// Datatypes/Structs/_TcVnKeyPoint
{attribute 'linkalways'} 
{attribute 'no_explicit_call' := 'This FB is a CLASS and must be accessed using methods or properties'}
{attribute 'enable_dynamic_creation'}
FUNCTION_BLOCK _TcVnKeyPoint EXTENDS StructuredDatatypeBase
VAR
	localData : TcVnKeyPoint;
	activeData : REFERENCE TO TcVnKeyPoint REF= localData;
    _aPoint : _TcVnPoint2_REAL();
    _fDiameter : _REAL(localdata.fDiameter);
    _fAngle : _REAL(localdata.fAngle);
    _fResponse : _REAL(localdata.fResponse);
    _nOctave : _DINT(localdata.nOctave);
    _nClassId : _DINT(localdata.nClassId);
END_VAR

PROPERTY PUBLIC Address : PVOID
GET
Address := ADR(activeData);
END_GET
END_PROPERTY

METHOD PUBLIC ClearReference
VAR_INPUT
END_VAR
activeData REF= localData;
SetMemberReference();
END_METHOD

PROPERTY PUBLIC Size : UDINT
GET
Size := SIZEOF(activeData);
END_GET
END_PROPERTY

METHOD FB_init : BOOL
VAR_INPUT
	bInitRetains : BOOL; // if TRUE, the retain variables are initialized (warm start / cold start)
	bInCopyCode : BOOL;  // if TRUE, the instance afterwards gets moved into the copy code (online change)
END_VAR
SetMemberReference();
AddMember('aPoint', _aPoint);
AddMember('fDiameter', _fDiameter);
AddMember('fAngle', _fAngle);
AddMember('fResponse', _fResponse);
AddMember('nOctave', _nOctave);
AddMember('nClassId', _nClassId);
END_METHOD

METHOD PROTECTED SetMemberReference
VAR_INPUT
END_VAR
_aPoint.MakeReferenceTo(activeData.aPoint);
_fDiameter.MakeReferenceTo(activeData.fDiameter);
_fAngle.MakeReferenceTo(activeData.fAngle);
_fResponse.MakeReferenceTo(activeData.fResponse);
_nOctave.MakeReferenceTo(activeData.nOctave);
_nClassId.MakeReferenceTo(activeData.nClassId);
END_METHOD

METHOD PUBLIC Clone : I_Datatype
VAR
    pClone : POINTER TO _TcVnKeyPoint;
END_VAR
pClone := __NEW(_TcVnKeyPoint());
pClone^.Value := Value;
Clone := pClone^;
END_METHOD

PROPERTY PUBLIC Identifier : T_MAXSTRING
GET
Identifier := 'TcVnKeyPoint';
END_GET
END_PROPERTY

METHOD PUBLIC MakeReferenceTo
VAR_INPUT
	ReferenceTarget : REFERENCE TO TcVnKeyPoint;
END_VAR
activeData REF= ReferenceTarget;
SetMemberReference();
END_METHOD

METHOD TryMakeReferenceTo : BOOL
VAR_INPUT
	Target : I_Datatype;
END_VAR
VAR
	pTargetData : POINTER TO TcVnKeyPoint;
END_VAR
IF NOT IsEquivalentTo(Target) THEN
	RETURN;
END_IF

pTargetData := Target.Address;
activeData REF= pTargetData^;
SetMemberReference();
TryMakeReferenceTo := TRUE;
END_METHOD

PROPERTY PUBLIC Value : REFERENCE TO TcVnKeyPoint
GET
Value REF= activeData;
END_GET
END_PROPERTY

PROPERTY PUBLIC aPoint : REFERENCE TO _TcVnPoint2_REAL
GET
aPoint REF= _aPoint;
END_GET
END_PROPERTY

PROPERTY PUBLIC fAngle : REFERENCE TO _REAL
GET
fAngle REF= _fAngle;
END_GET
END_PROPERTY

PROPERTY PUBLIC fDiameter : REFERENCE TO _REAL
GET
fDiameter REF= _fDiameter;
END_GET
END_PROPERTY

PROPERTY PUBLIC fResponse : REFERENCE TO _REAL
GET
fResponse REF= _fResponse;
END_GET
END_PROPERTY

PROPERTY PUBLIC nClassId : REFERENCE TO _DINT
GET
nClassId REF= _nClassId;
END_GET
END_PROPERTY

PROPERTY PUBLIC nOctave : REFERENCE TO _DINT
GET
nOctave REF= _nOctave;
END_GET
END_PROPERTY

END_FUNCTION_BLOCK

// Datatypes/Structs/_TcVnRotatedRectangle
{attribute 'linkalways'} 
{attribute 'no_explicit_call' := 'This FB is a CLASS and must be accessed using methods or properties'}
{attribute 'enable_dynamic_creation'}
FUNCTION_BLOCK _TcVnRotatedRectangle EXTENDS StructuredDatatypeBase
VAR
	localData : TcVnRotatedRectangle;
	activeData : REFERENCE TO TcVnRotatedRectangle REF= localData;
    _aCenter : _TcVnPoint2_REAL();
    _stSize : _TcVnSize2_REAL();
    _fAngle : _REAL(localdata.fAngle);
END_VAR

PROPERTY PUBLIC Address : PVOID
GET
Address := ADR(activeData);
END_GET
END_PROPERTY

METHOD PUBLIC ClearReference
VAR_INPUT
END_VAR
activeData REF= localData;
SetMemberReference();
END_METHOD

PROPERTY PUBLIC Size : UDINT
GET
Size := SIZEOF(activeData);
END_GET
END_PROPERTY

METHOD FB_init : BOOL
VAR_INPUT
	bInitRetains : BOOL; // if TRUE, the retain variables are initialized (warm start / cold start)
	bInCopyCode : BOOL;  // if TRUE, the instance afterwards gets moved into the copy code (online change)
END_VAR
SetMemberReference();
AddMember('aCenter', _aCenter);
AddMember('stSize', _stSize);
AddMember('fAngle', _fAngle);
END_METHOD

METHOD PROTECTED SetMemberReference
VAR_INPUT
END_VAR
_aCenter.MakeReferenceTo(activeData.aCenter);
_stsize.MakeReferenceTo(activeData.stSize);
_fAngle.MakeReferenceTo(activeData.fAngle);
END_METHOD

METHOD PUBLIC Clone : I_Datatype
VAR
    pClone : POINTER TO _TcVnRotatedRectangle;
END_VAR
pClone := __NEW(_TcVnRotatedRectangle());
pClone^.Value := Value;
Clone := pClone^;
END_METHOD

PROPERTY PUBLIC Identifier : T_MAXSTRING
GET
Identifier := 'TcVnRotatedRectangle';
END_GET
END_PROPERTY

METHOD PUBLIC MakeReferenceTo
VAR_INPUT
	ReferenceTarget : REFERENCE TO TcVnRotatedRectangle;
END_VAR
activeData REF= ReferenceTarget;
SetMemberReference();
END_METHOD

METHOD TryMakeReferenceTo : BOOL
VAR_INPUT
	Target : I_Datatype;
END_VAR
VAR
	pTargetData : POINTER TO TcVnRotatedRectangle;
END_VAR
IF NOT IsEquivalentTo(Target) THEN
	RETURN;
END_IF

pTargetData := Target.Address;
activeData REF= pTargetData^;
SetMemberReference();
TryMakeReferenceTo := TRUE;
END_METHOD

PROPERTY PUBLIC Value : REFERENCE TO TcVnRotatedRectangle
GET
Value REF= activeData;
END_GET
END_PROPERTY

PROPERTY PUBLIC aCenter : REFERENCE TO _TcVnPoint2_REAL
GET
aCenter REF= _aCenter;
END_GET
END_PROPERTY

PROPERTY PUBLIC fAngle : REFERENCE TO _REAL
GET
fAngle REF= _fAngle;
END_GET
END_PROPERTY

PROPERTY PUBLIC stSize : REFERENCE TO _TcVnSize2_REAL
GET
stSize REF= _stSize;
END_GET
END_PROPERTY

END_FUNCTION_BLOCK

// Datatypes/Structs/_TcVnSize2_REAL
{attribute 'linkalways'} 
{attribute 'no_explicit_call' := 'This FB is a CLASS and must be accessed using methods or properties'}
{attribute 'enable_dynamic_creation'}
FUNCTION_BLOCK _TcVnSize2_REAL EXTENDS StructuredDatatypeBase
VAR
	localData : TcVnSize2_REAL;
	activeData : REFERENCE TO TcVnSize2_REAL REF= localData;
    _fWidth : _REAL(localdata.fWidth);
    _fHeight : _REAL(localdata.fHeight);
END_VAR

PROPERTY PUBLIC Address : PVOID
GET
Address := ADR(activeData);
END_GET
END_PROPERTY

METHOD PUBLIC ClearReference
VAR_INPUT
END_VAR
activeData REF= localData;
SetMemberReference();
END_METHOD

PROPERTY PUBLIC Size : UDINT
GET
Size := SIZEOF(activeData);
END_GET
END_PROPERTY

METHOD FB_init : BOOL
VAR_INPUT
	bInitRetains : BOOL; // if TRUE, the retain variables are initialized (warm start / cold start)
	bInCopyCode : BOOL;  // if TRUE, the instance afterwards gets moved into the copy code (online change)
END_VAR
SetMemberReference();
AddMember('fWidth', _fWidth);
AddMember('fHeight', _fHeight);
END_METHOD

METHOD PROTECTED SetMemberReference
VAR_INPUT
END_VAR
_fWidth.MakeReferenceTo(activeData.fWidth);
_fHeight.MakeReferenceTo(activeData.fHeight);
END_METHOD

METHOD PUBLIC Clone : I_Datatype
VAR
    pClone : POINTER TO _TcVnSize2_REAL;
END_VAR
pClone := __NEW(_TcVnSize2_REAL());
pClone^.Value := Value;
Clone := pClone^;
END_METHOD

PROPERTY PUBLIC Identifier : T_MAXSTRING
GET
Identifier := 'TcVnSize2_REAL';
END_GET
END_PROPERTY

METHOD PUBLIC MakeReferenceTo
VAR_INPUT
	ReferenceTarget : REFERENCE TO TcVnSize2_REAL;
END_VAR
activeData REF= ReferenceTarget;
SetMemberReference();
END_METHOD

METHOD TryMakeReferenceTo : BOOL
VAR_INPUT
	Target : I_Datatype;
END_VAR
VAR
	pTargetData : POINTER TO TcVnSize2_REAL;
END_VAR
IF NOT IsEquivalentTo(Target) THEN
	RETURN;
END_IF

pTargetData := Target.Address;
activeData REF= pTargetData^;
SetMemberReference();
TryMakeReferenceTo := TRUE;
END_METHOD

PROPERTY PUBLIC Value : REFERENCE TO TcVnSize2_REAL
GET
Value REF= activeData;
END_GET
END_PROPERTY

PROPERTY PUBLIC fHeight : REFERENCE TO _REAL
GET
fHeight REF= _fHeight;
END_GET
END_PROPERTY

PROPERTY PUBLIC fWidth : REFERENCE TO _REAL
GET
fWidth REF= _fWidth;
END_GET
END_PROPERTY

END_FUNCTION_BLOCK

// Datatypes/Interfaces/Containers/Iterators/ITcVnBidirectionalIterator/_ITcVnBidirectionalIterator
{attribute 'linkalways'} 
{attribute 'no_explicit_call' := 'This FB is a CLASS and must be accessed using methods or properties'}
{attribute 'enable_dynamic_creation'}
FUNCTION_BLOCK _ITcVnBidirectionalIterator EXTENDS InterfaceDatatypeBase IMPLEMENTS I_InterfaceDatatype_ITcVnBidirectionalIterator
VAR
	localData : ITcVnBidirectionalIterator;
	activeData : REFERENCE TO ITcVnBidirectionalIterator REF= localData;
END_VAR

PROPERTY PUBLIC Address : PVOID
GET
Address := ADR(activeData);
END_GET
END_PROPERTY

METHOD PUBLIC ClearReference
VAR_INPUT
END_VAR
activeData REF= localData;
END_METHOD

PROPERTY PUBLIC Size : UDINT
GET
Size := SIZEOF(activeData);
END_GET
END_PROPERTY

METHOD FB_exit : BOOL
VAR_INPUT
	bInCopyCode : BOOL; // if TRUE, the exit method is called for exiting an instance that is copied afterwards (online change).
END_VAR
IF bInCopyCode THEN
	RETURN;
END_IF

TryTcReleaseLocal();
END_METHOD

METHOD PUBLIC TryTcReleaseLocal : BOOL
VAR_INPUT
END_VAR
IF localData = 0 THEN
	RETURN;
END_IF

IF localData.TcRelease() = 0 THEN
	localData := 0;
END_IF

TryTcReleaseLocal := TRUE;
END_METHOD

METHOD PUBLIC Clone : I_Datatype
VAR
    pClone : POINTER TO _ITcVnBidirectionalIterator;
END_VAR
pClone := __NEW(_ITcVnBidirectionalIterator);
Clone := pClone^;
END_METHOD

PROPERTY PUBLIC Identifier : T_MAXSTRING
GET
Identifier := 'ITcVnBidirectionalIterator';
END_GET
END_PROPERTY

METHOD PUBLIC MakeReferenceTo
VAR_INPUT
	ReferenceTarget : REFERENCE TO ITcVnBidirectionalIterator;
END_VAR
activeData REF= ReferenceTarget;
END_METHOD

METHOD PUBLIC SerializeWith
VAR_INPUT
	Serializer : I_Serializer;
END_VAR
Serializer.AddNull();
END_METHOD

METHOD TryDeserializeFrom : BOOL
VAR_INPUT
	Deserializer : I_Deserializer;
	Feedback : I_DeserializerFeedback;
END_VAR
VAR
END_VAR
// not implemented.
END_METHOD

METHOD TryMakeReferenceTo : BOOL
VAR_INPUT
	Target : I_Datatype;
END_VAR
VAR
	pTargetData : POINTER TO ITcVnBidirectionalIterator;
END_VAR
IF NOT IsEquivalentTo(Target) THEN
	RETURN;
END_IF

pTargetData := Target.Address;
activeData REF= pTargetData^;
TryMakeReferenceTo := TRUE;
END_METHOD

PROPERTY PUBLIC Value : REFERENCE TO ITcVnBidirectionalIterator
GET
Value REF= activeData;
END_GET
END_PROPERTY

PROPERTY PUBLIC IsValid : BOOL
GET
IsValid := activeData <> 0;
END_GET
END_PROPERTY

METHOD PUBLIC TryCheckIfBegin : BOOL
VAR_INPUT
	Result : REFERENCE TO BOOL;
END_VAR
Result := FALSE;

IF NOT IsValid THEN
	RETURN;
END_IF

IF activeData.CheckIfBegin() = S_OK THEN
    Result := TRUE;
END_IF

TryCheckIfBegin := TRUE;
END_METHOD

METHOD PUBLIC TryCheckIfEnd : BOOL
VAR_INPUT
	Result : REFERENCE TO BOOL;
END_VAR
Result := FALSE;

IF NOT IsValid THEN
	RETURN;
END_IF

IF activeData.CheckIfEnd() = S_OK THEN
    Result := TRUE;
END_IF

TryCheckIfEnd := TRUE;
END_METHOD

METHOD PUBLIC TryCopyContentFrom : BOOL
VAR_INPUT
	Source : I_InterfaceDatatype;
END_VAR
// currently un-copyable
END_METHOD

METHOD PUBLIC TryGetValueSize : BOOL
VAR_INPUT
	Destination : REFERENCE TO ULINT;
END_VAR
IF NOT IsValid THEN
	RETURN;
END_IF

TryGetValueSize := SUCCEEDED(activeData.GetValueSize(Destination));
END_METHOD

METHOD PUBLIC TryGetValueTypeGuid : BOOL
VAR_INPUT
	Destination : REFERENCE TO GUID;
END_VAR
IF NOT IsValid THEN
	RETURN;
END_IF

TryGetValueTypeGuid := SUCCEEDED(activeData.GetValueTypeGuid(Destination));
END_METHOD

METHOD PUBLIC TryTcAddRef : BOOL
VAR_INPUT
END_VAR
IF activeData = 0 THEN
	RETURN;
END_IF

IF activeData.TcAddRef() = 0 THEN
	activeData := 0;
END_IF

TryTcAddRef := TRUE;
END_METHOD

METHOD PUBLIC TryTcRelease : BOOL
VAR_INPUT
END_VAR
IF activeData = 0 THEN
	RETURN;
END_IF

IF activeData.TcRelease() = 0 THEN
	activeData := 0;
END_IF

TryTcRelease := TRUE;
END_METHOD

END_FUNCTION_BLOCK

// Datatypes/Interfaces/Containers/Iterators/ITcVnBidirectionalIterator/I_InterfaceDatatype_ITcVnBidirectionalIterator
INTERFACE I_InterfaceDatatype_ITcVnBidirectionalIterator EXTENDS I_InterfaceDatatype

PROPERTY PUBLIC Value : REFERENCE TO ITcVnBidirectionalIterator
GET
END_GET
END_PROPERTY

END_INTERFACE

// Datatypes/Interfaces/Images/ITcVnDisplayableImage/_ITcVnDisplayableImage
{attribute 'linkalways'} 
{attribute 'no_explicit_call' := 'This FB is a CLASS and must be accessed using methods or properties'}
{attribute 'enable_dynamic_creation'}
FUNCTION_BLOCK _ITcVnDisplayableImage EXTENDS InterfaceDatatypeBase IMPLEMENTS I_InterfaceDatatype_ITcVnDisplayableImage
VAR
	localData : ITcVnDisplayableImage;
	activeData : REFERENCE TO ITcVnDisplayableImage REF= localData;
END_VAR

PROPERTY PUBLIC Address : PVOID
GET
Address := ADR(activeData);
END_GET
END_PROPERTY

METHOD PUBLIC ClearReference
VAR_INPUT
END_VAR
activeData REF= localData;
END_METHOD

PROPERTY PUBLIC Size : UDINT
GET
Size := SIZEOF(activeData);
END_GET
END_PROPERTY

METHOD FB_exit : BOOL
VAR_INPUT
	bInCopyCode : BOOL; // if TRUE, the exit method is called for exiting an instance that is copied afterwards (online change).
END_VAR
IF bInCopyCode THEN
	RETURN;
END_IF

TryTcReleaseLocal();
END_METHOD

METHOD PUBLIC TryTcReleaseLocal : BOOL
VAR_INPUT
END_VAR
IF localData = 0 THEN
	RETURN;
END_IF

IF localData.TcRelease() = 0 THEN
	localData := 0;
END_IF

TryTcReleaseLocal := TRUE;
END_METHOD

METHOD PUBLIC Clone : I_Datatype
VAR
    pClone : POINTER TO _ITcVnDisplayableImage;
END_VAR
pClone := __NEW(_ITcVnDisplayableImage);
Clone := pClone^;
END_METHOD

PROPERTY PUBLIC Identifier : T_MAXSTRING
GET
Identifier := 'ITcVnDisplayableImage';
END_GET
END_PROPERTY

METHOD PUBLIC MakeReferenceTo
VAR_INPUT
	ReferenceTarget : REFERENCE TO ITcVnDisplayableImage;
END_VAR
activeData REF= ReferenceTarget;
END_METHOD

METHOD PUBLIC SerializeWith
VAR_INPUT
	Serializer : I_Serializer;
END_VAR
// not possible to serialize the data.
Serializer.AddNull();
END_METHOD

METHOD TryMakeReferenceTo : BOOL
VAR_INPUT
	Target : I_Datatype;
END_VAR
VAR
	pTargetData : POINTER TO ITcVnDisplayableImage;
END_VAR
IF NOT IsEquivalentTo(Target) THEN
	RETURN;
END_IF

pTargetData := Target.Address;
activeData REF= pTargetData^;
TryMakeReferenceTo := TRUE;
END_METHOD

PROPERTY PUBLIC Value : REFERENCE TO ITcVnDisplayableImage
GET
Value REF= activeData;
END_GET
END_PROPERTY

PROPERTY PUBLIC IsValid : BOOL
GET
IsValid := activeData <> 0;
END_GET
END_PROPERTY

METHOD PUBLIC TryCopyContentFrom : BOOL
VAR_INPUT
	Source : I_InterfaceDatatype;
END_VAR
// not possible to copy the data, so this will always fail
END_METHOD

METHOD TryDeserializeFrom : BOOL
VAR_INPUT
	Deserializer : I_Deserializer;
	Feedback : I_DeserializerFeedback;
END_VAR
// not possible to deserialize from data.
TryDeserializeFrom := TRUE;
END_METHOD

METHOD PUBLIC TryTcAddRef : BOOL
VAR_INPUT
END_VAR
IF activeData = 0 THEN
	RETURN;
END_IF

IF activeData.TcAddRef() = 0 THEN
	activeData := 0;
END_IF

TryTcAddRef := TRUE;
END_METHOD

METHOD PUBLIC TryTcRelease : BOOL
VAR_INPUT
END_VAR
IF activeData = 0 THEN
	RETURN;
END_IF

IF activeData.TcRelease() = 0 THEN
	activeData := 0;
END_IF

TryTcRelease := TRUE;
END_METHOD

END_FUNCTION_BLOCK

// Datatypes/Interfaces/Images/ITcVnDisplayableImage/I_InterfaceDatatype_ITcVnDisplayableImage
INTERFACE I_InterfaceDatatype_ITcVnDisplayableImage EXTENDS I_InterfaceDatatype

PROPERTY PUBLIC Value : REFERENCE TO ITcVnDisplayableImage
GET
END_GET
END_PROPERTY

END_INTERFACE

// Datatypes/Structs/_GVCP_ADDRESS_VALUE_PAIR
{attribute 'linkalways'}
{attribute 'no_explicit_call' := 'This FB is a CLASS and must be accessed using methods or properties'}
{attribute 'enable_dynamic_creation'}
FUNCTION_BLOCK _GVCP_ADDRESS_VALUE_PAIR EXTENDS StructuredDatatypeBase
VAR
    localData : GVCP_ADDRESS_VALUE_PAIR;
    activeData : REFERENCE TO GVCP_ADDRESS_VALUE_PAIR REF= localData;
    _nAddress : _GVCP_REGISTER_ADDRESS(0);
    _nValue : _GVCP_REGISTER_VALUE(0);
END_VAR

PROPERTY PUBLIC Address : PVOID
GET
Address := ADR(activeData);
END_GET
END_PROPERTY

METHOD PUBLIC ClearReference
VAR_INPUT
END_VAR
activeData REF= localData;
SetMemberReference();
END_METHOD

PROPERTY PUBLIC Size : UDINT
GET
Size := SIZEOF(activeData);
END_GET
END_PROPERTY

METHOD FB_init : BOOL
VAR_INPUT
	bInitRetains : BOOL; // if TRUE, the retain variables are initialized (warm start / cold start)
	bInCopyCode : BOOL;  // if TRUE, the instance afterwards gets moved into the copy code (online change)
END_VAR
SetMemberReference();
AddMember('nAddress', _nAddress);
AddMember('nValue', _nValue);
END_METHOD

METHOD PROTECTED SetMemberReference
VAR_INPUT
END_VAR
_nAddress.MakeReferenceTo(activeData.nAddress);
_nValue.MakeReferenceTo(activeData.nValue);
END_METHOD

METHOD PUBLIC Clone : I_Datatype
VAR
    pClone : POINTER TO _GVCP_ADDRESS_VALUE_PAIR;
END_VAR
pClone := __NEW(_GVCP_ADDRESS_VALUE_PAIR);
IF pClone = 0 THEN
    RETURN;
END_IF
pClone^.TryCopyFrom(THIS^);
Clone := pClone^;
END_METHOD

PROPERTY PUBLIC Identifier : T_MAXSTRING
GET
Identifier := 'GVCP_ADDRESS_VALUE_PAIR';
END_GET
END_PROPERTY

METHOD PUBLIC MakeReferenceTo
VAR_INPUT
	ReferenceTarget : REFERENCE TO GVCP_ADDRESS_VALUE_PAIR;
END_VAR
activeData REF= ReferenceTarget;
SetMemberReference();
END_METHOD

METHOD TryMakeReferenceTo : BOOL
VAR_INPUT
	Target : I_Datatype;
END_VAR
VAR
	pTargetData : POINTER TO GVCP_ADDRESS_VALUE_PAIR;
END_VAR
IF NOT IsEquivalentTo(Target) THEN
	RETURN;
END_IF

pTargetData := Target.Address;
activeData REF= pTargetData^;
SetMemberReference();
TryMakeReferenceTo := TRUE;
END_METHOD

PROPERTY PUBLIC Value : REFERENCE TO GVCP_ADDRESS_VALUE_PAIR
GET
Value REF= activeData;
END_GET
END_PROPERTY

PROPERTY PUBLIC nAddress : REFERENCE TO _GVCP_REGISTER_ADDRESS
GET
nAddress REF= _nAddress;
END_GET
END_PROPERTY

PROPERTY PUBLIC nValue : REFERENCE TO _GVCP_REGISTER_VALUE
GET
nValue REF= _nValue;
END_GET
END_PROPERTY

END_FUNCTION_BLOCK

// Datatypes/Structs/_GVSP_IMAGE_INFO
{attribute 'linkalways'} 
{attribute 'no_explicit_call' := 'This FB is a CLASS and must be accessed using methods or properties'}
{attribute 'enable_dynamic_creation'}
FUNCTION_BLOCK _GVSP_IMAGE_INFO EXTENDS StructuredDatatypeBase
VAR
	localData : GVSP_IMAGE_INFO;
	activeData : REFERENCE TO GVSP_IMAGE_INFO REF= localData;
    _CameraIpAddress : _UDINT(localdata.CameraIpAddress);
    _LocalIpAddress : _UDINT(localdata.LocalIpAddress);
    _CameraUdpPort : _UINT(localdata.CameraUdpPort);
    _LocalUdpPort : _UINT(localdata.LocalUdpPort);
    _GvspChannelId : _UINT(localdata.GvspChannelId);
    _GevStatus : _UINT(localdata.GevStatus);
    _BlockId : _ULINT(localdata.BlockId);
    _LeaderInfo : _GVSP_LEADER_PAYLOAD_IMAGE();
END_VAR

PROPERTY PUBLIC Address : PVOID
GET
Address := ADR(activeData);
END_GET
END_PROPERTY

METHOD PUBLIC ClearReference
VAR_INPUT
END_VAR
activeData REF= localData;
SetMemberReference();
END_METHOD

PROPERTY PUBLIC Size : UDINT
GET
Size := SIZEOF(activeData);
END_GET
END_PROPERTY

METHOD FB_init : BOOL
VAR_INPUT
	bInitRetains : BOOL; // if TRUE, the retain variables are initialized (warm start / cold start)
	bInCopyCode : BOOL;  // if TRUE, the instance afterwards gets moved into the copy code (online change)
END_VAR
SetMemberReference();
AddMember('CameraIpAddress', _CameraIpAddress);
AddMember('LocalIpAddress', _LocalIpAddress);
AddMember('CameraUdpPort', _CameraUdpPort);
AddMember('LocalUdpPort', _LocalUdpPort);
AddMember('GvspChannelId', _GvspChannelId);
AddMember('GevStatus', _GevStatus);
AddMember('BlockId', _BlockId);
AddMember('LeaderInfo', _LeaderInfo);
END_METHOD

METHOD PROTECTED SetMemberReference
VAR_INPUT
END_VAR
_CameraIpAddress.MakeReferenceTo(activeData.CameraIpAddress);
_LocalIpAddress.MakeReferenceTo(activeData.LocalIpAddress);
_CameraUdpPort.MakeReferenceTo(activeData.CameraUdpPort);
_LocalUdpPort.MakeReferenceTo(activeData.LocalUdpPort);
_GvspChannelId.MakeReferenceTo(activeData.GvspChannelId);
_GevStatus.MakeReferenceTo(activeData.GevStatus);
_BlockId.MakeReferenceTo(activeData.BlockId);
_LeaderInfo.MakeReferenceTo(activeData.LeaderInfo);
END_METHOD

METHOD PUBLIC Clone : I_Datatype
VAR
    pClone : POINTER TO _GVSP_IMAGE_INFO;
END_VAR
pClone := __NEW(_GVSP_IMAGE_INFO());
pClone^.Value := Value;
Clone := pClone^;
END_METHOD

PROPERTY PUBLIC Identifier : T_MAXSTRING
GET
Identifier := 'GVSP_IMAGE_INFO';
END_GET
END_PROPERTY

METHOD PUBLIC MakeReferenceTo
VAR_INPUT
	ReferenceTarget : REFERENCE TO GVSP_IMAGE_INFO;
END_VAR
activeData REF= ReferenceTarget;
SetMemberReference();
END_METHOD

METHOD TryMakeReferenceTo : BOOL
VAR_INPUT
	Target : I_Datatype;
END_VAR
VAR
	targetAsStruct : I_StructuredDatatype;
	pTargetData : POINTER TO GVSP_IMAGE_INFO;
END_VAR
IF NOT Target.TryResolveAsStructuredDatatype(targetAsStruct) THEN
	RETURN;
END_IF

IF NOT (targetAsStruct.Identifier = Identifier) THEN
	RETURN;
END_IF

pTargetData := Target.Address;
activeData REF= pTargetData^;
SetMemberReference();
TryMakeReferenceTo := TRUE;
END_METHOD

PROPERTY PUBLIC Value : REFERENCE TO GVSP_IMAGE_INFO
GET
Value REF= activeData;
END_GET
END_PROPERTY

PROPERTY PUBLIC BlockId : REFERENCE TO _ULINT
GET
BlockId REF= _BlockId;
END_GET
END_PROPERTY

PROPERTY PUBLIC CameraIpAddress : REFERENCE TO _UDINT
GET
CameraIpAddress REF= _CameraIpAddress;
END_GET
END_PROPERTY

PROPERTY PUBLIC CameraUdpPort : REFERENCE TO _UINT
GET
CameraUdpPort REF= _CameraUdpPort;
END_GET
END_PROPERTY

PROPERTY PUBLIC GevStatus : REFERENCE TO _UINT
GET
GevStatus REF= _GevStatus;
END_GET
END_PROPERTY

PROPERTY PUBLIC GvspChannelId : REFERENCE TO _UINT
GET
GvspChannelId REF= _GvspChannelId;
END_GET
END_PROPERTY

PROPERTY PUBLIC LeaderInfo : REFERENCE TO _GVSP_LEADER_PAYLOAD_IMAGE
GET
LeaderInfo REF= _LeaderInfo;
END_GET
END_PROPERTY

PROPERTY PUBLIC LocalIpAddress : REFERENCE TO _UDINT
GET
LocalIpAddress REF= _LocalIpAddress;
END_GET
END_PROPERTY

PROPERTY PUBLIC LocalUdpPort : REFERENCE TO _UINT
GET
LocalUdpPort REF= _LocalUdpPort;
END_GET
END_PROPERTY

END_FUNCTION_BLOCK

// Datatypes/Structs/_GVSP_LEADER_PAYLOAD_IMAGE
{attribute 'linkalways'} 
{attribute 'no_explicit_call' := 'This FB is a CLASS and must be accessed using methods or properties'}
{attribute 'enable_dynamic_creation'}
FUNCTION_BLOCK _GVSP_LEADER_PAYLOAD_IMAGE EXTENDS StructuredDatatypeBase
VAR
	localData : GVSP_LEADER_PAYLOAD_IMAGE;
	activeData : REFERENCE TO GVSP_LEADER_PAYLOAD_IMAGE REF= localData;
    _Timestamp : _ULINT(localdata.Timestamp);
    _PixelFormat : _GVSP_PIXEL_FORMAT();
    _SizeX : _UDINT(localdata.SizeX);
    _SizeY : _UDINT(localdata.SizeY);
    _OffsetX : _UDINT(localdata.OffsetX);
    _OffsetY : _UDINT(localdata.OffsetY);
    _PaddingX : _UINT(localdata.PaddingX);
    _PaddingY : _UINT(localdata.PaddingY);
END_VAR

PROPERTY PUBLIC Address : PVOID
GET
Address := ADR(activeData);
END_GET
END_PROPERTY

METHOD PUBLIC ClearReference
VAR_INPUT
END_VAR
activeData REF= localData;
SetMemberReference();
END_METHOD

PROPERTY PUBLIC Size : UDINT
GET
Size := SIZEOF(activeData);
END_GET
END_PROPERTY

METHOD FB_init : BOOL
VAR_INPUT
	bInitRetains : BOOL; // if TRUE, the retain variables are initialized (warm start / cold start)
	bInCopyCode : BOOL;  // if TRUE, the instance afterwards gets moved into the copy code (online change)
END_VAR
SetMemberReference();
AddMember('Timestamp', _Timestamp);
AddMember('PixelFormat', _PixelFormat);
AddMember('SizeX', _SizeX);
AddMember('SizeY', _SizeY);
AddMember('OffsetX', _OffsetX);
AddMember('OffsetY', _OffsetY);
AddMember('PaddingX', _PaddingX);
AddMember('PaddingY', _PaddingY);
END_METHOD

METHOD PROTECTED SetMemberReference
VAR_INPUT
END_VAR
_Timestamp.MakeReferenceTo(activeData.Timestamp);
_PixelFormat.MakeReferenceTo(activeData.PixelFormat);
_SizeX.MakeReferenceTo(activeData.SizeX);
_SizeY.MakeReferenceTo(activeData.SizeY);
_OffsetX.MakeReferenceTo(activeData.OffsetX);
_OffsetY.MakeReferenceTo(activeData.OffsetY);
_PaddingX.MakeReferenceTo(activeData.PaddingX);
_PaddingY.MakeReferenceTo(activeData.PaddingY);
END_METHOD

METHOD PUBLIC Clone : I_Datatype
VAR
    pClone : POINTER TO _GVSP_LEADER_PAYLOAD_IMAGE;
END_VAR
pClone := __NEW(_GVSP_LEADER_PAYLOAD_IMAGE());
pClone^.Value := Value;
Clone := pClone^;
END_METHOD

PROPERTY PUBLIC Identifier : T_MAXSTRING
GET
Identifier := 'GVSP_LEADER_PAYLOAD_IMAGE';
END_GET
END_PROPERTY

METHOD PUBLIC MakeReferenceTo
VAR_INPUT
	ReferenceTarget : REFERENCE TO GVSP_LEADER_PAYLOAD_IMAGE;
END_VAR
activeData REF= ReferenceTarget;
SetMemberReference();
END_METHOD

METHOD TryMakeReferenceTo : BOOL
VAR_INPUT
	Target : I_Datatype;
END_VAR
VAR
	targetAsStruct : I_StructuredDatatype;
	pTargetData : POINTER TO GVSP_LEADER_PAYLOAD_IMAGE;
END_VAR
IF NOT Target.TryResolveAsStructuredDatatype(targetAsStruct) THEN
	RETURN;
END_IF

IF NOT (targetAsStruct.Identifier = Identifier) THEN
	RETURN;
END_IF

pTargetData := Target.Address;
activeData REF= pTargetData^;
SetMemberReference();
TryMakeReferenceTo := TRUE;
END_METHOD

PROPERTY PUBLIC Value : REFERENCE TO GVSP_LEADER_PAYLOAD_IMAGE
GET
Value REF= activeData;
END_GET
END_PROPERTY

PROPERTY PUBLIC OffsetX : REFERENCE TO _UDINT
GET
OffsetX REF= _OffsetX;
END_GET
END_PROPERTY

PROPERTY PUBLIC OffsetY : REFERENCE TO _UDINT
GET
OffsetY REF= _OffsetY;
END_GET
END_PROPERTY

PROPERTY PUBLIC PaddingX : REFERENCE TO _UINT
GET
PaddingX REF= _PaddingX;
END_GET
END_PROPERTY

PROPERTY PUBLIC PaddingY : REFERENCE TO _UINT
GET
PaddingY REF= _PaddingY;
END_GET
END_PROPERTY

PROPERTY PUBLIC PixelFormat : REFERENCE TO _GVSP_PIXEL_FORMAT
GET
PixelFormat REF= _PixelFormat;
END_GET
END_PROPERTY

PROPERTY PUBLIC SizeX : REFERENCE TO _UDINT
GET
SizeX REF= _SizeX;
END_GET
END_PROPERTY

PROPERTY PUBLIC SizeY : REFERENCE TO _UDINT
GET
SizeY REF= _SizeY;
END_GET
END_PROPERTY

PROPERTY PUBLIC Timestamp : REFERENCE TO _ULINT
GET
Timestamp REF= _Timestamp;
END_GET
END_PROPERTY

END_FUNCTION_BLOCK

// Datatypes/Structs/_GVSP_PIXEL_FORMAT
{attribute 'linkalways'} 
{attribute 'no_explicit_call' := 'This FB is a CLASS and must be accessed using methods or properties'}
{attribute 'enable_dynamic_creation'}
FUNCTION_BLOCK _GVSP_PIXEL_FORMAT EXTENDS StructuredDatatypeBase
VAR
	localData : GVSP_PIXEL_FORMAT;
	activeData : REFERENCE TO GVSP_PIXEL_FORMAT REF= localData;
    _Color : _BYTE(localdata.Color);
    _EffectivePixelSize : _BYTE(localdata.EffectivePixelSize);
    _Id : _UINT(localdata.Id);
END_VAR

PROPERTY PUBLIC Address : PVOID
GET
Address := ADR(activeData);
END_GET
END_PROPERTY

METHOD PUBLIC ClearReference
VAR_INPUT
END_VAR
activeData REF= localData;
SetMemberReference();
END_METHOD

PROPERTY PUBLIC Size : UDINT
GET
Size := SIZEOF(activeData);
END_GET
END_PROPERTY

METHOD FB_init : BOOL
VAR_INPUT
	bInitRetains : BOOL; // if TRUE, the retain variables are initialized (warm start / cold start)
	bInCopyCode : BOOL;  // if TRUE, the instance afterwards gets moved into the copy code (online change)
END_VAR
SetMemberReference();
AddMember('Color', _Color);
AddMember('EffectivePixelSize', _EffectivePixelSize);
AddMember('Id', _Id);
END_METHOD

METHOD PROTECTED SetMemberReference
VAR_INPUT
END_VAR
_Color.MakeReferenceTo(activeData.Color);
_EffectivePixelSize.MakeReferenceTo(activeData.EffectivePixelSize);
_Id.MakeReferenceTo(activeData.Id);
END_METHOD

METHOD PUBLIC Clone : I_Datatype
VAR
    pClone : POINTER TO _GVSP_PIXEL_FORMAT;
END_VAR
pClone := __NEW(_GVSP_PIXEL_FORMAT());
pClone^.Value := Value;
Clone := pClone^;
END_METHOD

PROPERTY PUBLIC Identifier : T_MAXSTRING
GET
Identifier := 'GVSP_PIXEL_FORMAT';
END_GET
END_PROPERTY

METHOD PUBLIC MakeReferenceTo
VAR_INPUT
	ReferenceTarget : REFERENCE TO GVSP_PIXEL_FORMAT;
END_VAR
activeData REF= ReferenceTarget;
SetMemberReference();
END_METHOD

METHOD TryMakeReferenceTo : BOOL
VAR_INPUT
	Target : I_Datatype;
END_VAR
VAR
	targetAsStruct : I_StructuredDatatype;
	pTargetData : POINTER TO GVSP_PIXEL_FORMAT;
END_VAR
IF NOT Target.TryResolveAsStructuredDatatype(targetAsStruct) THEN
	RETURN;
END_IF

IF NOT (targetAsStruct.Identifier = Identifier) THEN
	RETURN;
END_IF

pTargetData := Target.Address;
activeData REF= pTargetData^;
SetMemberReference();
TryMakeReferenceTo := TRUE;
END_METHOD

PROPERTY PUBLIC Value : REFERENCE TO GVSP_PIXEL_FORMAT
GET
Value REF= activeData;
END_GET
END_PROPERTY

PROPERTY PUBLIC Color : REFERENCE TO _BYTE
GET
Color REF= _Color;
END_GET
END_PROPERTY

PROPERTY PUBLIC EffectivePixelSize : REFERENCE TO _BYTE
GET
EffectivePixelSize REF= _EffectivePixelSize;
END_GET
END_PROPERTY

PROPERTY PUBLIC Id : REFERENCE TO _UINT
GET
Id REF= _Id;
END_GET
END_PROPERTY

END_FUNCTION_BLOCK

// Datatypes/Structs/_TcVnCameraCalibrationOptions
{attribute 'linkalways'} 
{attribute 'no_explicit_call' := 'This FB is a CLASS and must be accessed using methods or properties'}
{attribute 'enable_dynamic_creation'}
FUNCTION_BLOCK _TcVnCameraCalibrationOptions EXTENDS StructuredDatatypeBase
VAR
	localData : TcVnCameraCalibrationOptions;
	activeData : REFERENCE TO TcVnCameraCalibrationOptions REF= localData;

    _bUseIntrinsicGuess : _BIT();
    _bFixAspectRatio    : _BIT();
    _bFixPrincipalPoint : _BIT();
    _bZeroTangentDist   : _BIT();
    _bFixFocalLength    : _BIT();
    _bFixK1             : _BIT();
    _bFixK2             : _BIT();
    _bFixK3             : _BIT();
    _bFixK4             : _BIT();
    _bFixK5             : _BIT();
    _bFixK6             : _BIT();
    _bRationalModel     : _BIT();
END_VAR

PROPERTY PUBLIC Address : PVOID
GET
Address := ADR(activeData);
END_GET
END_PROPERTY

METHOD PUBLIC ClearReference
VAR_INPUT
END_VAR
activeData REF= localData;
SetMemberReference();
END_METHOD

PROPERTY PUBLIC Size : UDINT
GET
Size := SIZEOF(activeData);
END_GET
END_PROPERTY

METHOD FB_init : BOOL
VAR_INPUT
	bInitRetains : BOOL; // if TRUE, the retain variables are initialized (warm start / cold start)
	bInCopyCode : BOOL;  // if TRUE, the instance afterwards gets moved into the copy code (online change)
END_VAR
SetMemberReference();
AddMember('bUseIntrinsicGuess',_bUseIntrinsicGuess);
AddMember('bFixAspectRatio',_bFixAspectRatio);
AddMember('bFixPrincipalPoint',_bFixPrincipalPoint);
AddMember('bZeroTangentDist',_bZeroTangentDist);
AddMember('bFixFocalLength',_bFixFocalLength);
AddMember('bFixK1',_bFixK1);
AddMember('bFixK2',_bFixK2);
AddMember('bFixK3',_bFixK3);
AddMember('bFixK4',_bFixK4);
AddMember('bFixK5',_bFixK5);
AddMember('bFixK6',_bFixK6);
AddMember('bRationalModel',_bRationalModel);
END_METHOD

METHOD PROTECTED SetMemberReference
VAR_STAT
	// this variable is used for BITADR as this function fails if used on a local variable.
	structure : TcVnCameraCalibrationOptions;
END_VAR
_bUseIntrinsicGuess.MakeReferenceTo(THIS^, GetByteOffset(localData, localData.bUseIntrinsicGuess), BITADR(structure.bUseIntrinsicGuess));
_bFixAspectRatio.MakeReferenceTo(THIS^, GetByteOffset(localData, localData.bFixAspectRatio), BITADR(structure.bFixAspectRatio));
_bFixPrincipalPoint.MakeReferenceTo(THIS^, GetByteOffset(localData, localData.bFixPrincipalPoint), BITADR(structure.bFixPrincipalPoint));
_bZeroTangentDist.MakeReferenceTo(THIS^, GetByteOffset(localData, localData.bZeroTangentDist), BITADR(structure.bZeroTangentDist));
_bFixFocalLength.MakeReferenceTo(THIS^, GetByteOffset(localData, localData.bFixFocalLength), BITADR(structure.bFixFocalLength));
_bFixK1.MakeReferenceTo(THIS^, GetByteOffset(localData, localData.bFixK1), BITADR(structure.bFixK1));
_bFixK2.MakeReferenceTo(THIS^, GetByteOffset(localData, localData.bFixK2), BITADR(structure.bFixK2));
_bFixK3.MakeReferenceTo(THIS^, GetByteOffset(localData, localData.bFixK3), BITADR(structure.bFixK3));
_bFixK4.MakeReferenceTo(THIS^, GetByteOffset(localData, localData.bFixK4), BITADR(structure.bFixK4));
_bFixK5.MakeReferenceTo(THIS^, GetByteOffset(localData, localData.bFixK5), BITADR(structure.bFixK5));
_bFixK6.MakeReferenceTo(THIS^, GetByteOffset(localData, localData.bFixK6), BITADR(structure.bFixK6));
_bRationalModel.MakeReferenceTo(THIS^, GetByteOffset(localData, localData.bRationalModel), BITADR(structure.bRationalModel));
END_METHOD

METHOD PUBLIC Clone : I_Datatype
VAR
    pClone : POINTER TO _TcVnCameraCalibrationOptions;
END_VAR
pClone := __NEW(_TcVnCameraCalibrationOptions());
pClone^.Value := Value;
Clone := pClone^;
END_METHOD

PROPERTY PUBLIC Identifier : T_MAXSTRING
GET
Identifier := 'TcVnCameraCalibrationOptions';
END_GET
END_PROPERTY

METHOD PUBLIC MakeReferenceTo
VAR_INPUT
	ReferenceTarget : REFERENCE TO TcVnCameraCalibrationOptions;
END_VAR
activeData REF= ReferenceTarget;
SetMemberReference();
END_METHOD

METHOD TryMakeReferenceTo : BOOL
VAR_INPUT
	Target : I_Datatype;
END_VAR
VAR
	pTargetData : POINTER TO TcVnCameraCalibrationOptions;
END_VAR
IF NOT IsEquivalentTo(Target) THEN
	RETURN;
END_IF

pTargetData := Target.Address;
activeData REF= pTargetData^;
SetMemberReference();
TryMakeReferenceTo := TRUE;
END_METHOD

PROPERTY PUBLIC Value : REFERENCE TO TcVnCameraCalibrationOptions
GET
Value REF= activeData;
END_GET
END_PROPERTY

PROPERTY PUBLIC bFixAspectRatio : REFERENCE TO _BIT
GET
bFixAspectRatio REF= _bFixAspectRatio;
END_GET
END_PROPERTY

PROPERTY PUBLIC bFixFocalLength : REFERENCE TO _BIT
GET
bFixFocalLength REF= _bFixFocalLength;
END_GET
END_PROPERTY

PROPERTY PUBLIC bFixK1 : REFERENCE TO _BIT
GET
bFixK1 REF= _bFixK1;
END_GET
END_PROPERTY

PROPERTY PUBLIC bFixK2 : REFERENCE TO _BIT
GET
bFixK2 REF= _bFixK2;
END_GET
END_PROPERTY

PROPERTY PUBLIC bFixK3 : REFERENCE TO _BIT
GET
bFixK3 REF= _bFixK3;
END_GET
END_PROPERTY

PROPERTY PUBLIC bFixK4 : REFERENCE TO _BIT
GET
bFixK4 REF= _bFixK4;
END_GET
END_PROPERTY

PROPERTY PUBLIC bFixK5 : REFERENCE TO _BIT
GET
bFixK5 REF= _bFixK5;
END_GET
END_PROPERTY

PROPERTY PUBLIC bFixK6 : REFERENCE TO _BIT
GET
bFixK6 REF= _bFixK6;
END_GET
END_PROPERTY

PROPERTY PUBLIC bFixPrincipalPoint : REFERENCE TO _BIT
GET
bFixPrincipalPoint REF= _bFixPrincipalPoint;
END_GET
END_PROPERTY

PROPERTY PUBLIC bRationalModel : REFERENCE TO _BIT
GET
bRationalModel REF= _bRationalModel;
END_GET
END_PROPERTY

PROPERTY PUBLIC bUseIntrinsicGuess : REFERENCE TO _BIT
GET
bUseIntrinsicGuess REF= _bUseIntrinsicGuess;
END_GET
END_PROPERTY

PROPERTY PUBLIC bZeroTangentDist : REFERENCE TO _BIT
GET
bZeroTangentDist REF= _bZeroTangentDist;
END_GET
END_PROPERTY

END_FUNCTION_BLOCK

// Datatypes/Structs/_TcVnCircularArc
{attribute 'linkalways'} 
{attribute 'no_explicit_call' := 'This FB is a CLASS and must be accessed using methods or properties'}
{attribute 'enable_dynamic_creation'}
FUNCTION_BLOCK _TcVnCircularArc EXTENDS StructuredDatatypeBase
VAR
	localData : TcVnCircularArc;
	activeData : REFERENCE TO TcVnCircularArc REF= localData;
    _aCenter : _TcVnPoint2_REAL();
    _fRadius : _REAL(localdata.fRadius);
    _fStartAngle : _REAL(localdata.fStartAngle);
    _fEndAngle : _REAL(localdata.fEndAngle);
END_VAR

PROPERTY PUBLIC Address : PVOID
GET
Address := ADR(activeData);
END_GET
END_PROPERTY

METHOD PUBLIC ClearReference
VAR_INPUT
END_VAR
activeData REF= localData;
SetMemberReference();
END_METHOD

PROPERTY PUBLIC Size : UDINT
GET
Size := SIZEOF(activeData);
END_GET
END_PROPERTY

METHOD FB_init : BOOL
VAR_INPUT
	bInitRetains : BOOL; // if TRUE, the retain variables are initialized (warm start / cold start)
	bInCopyCode : BOOL;  // if TRUE, the instance afterwards gets moved into the copy code (online change)
END_VAR
SetMemberReference();
AddMember('aCenter', _aCenter);
AddMember('fRadius', _fRadius);
AddMember('fStartAngle', _fStartAngle);
AddMember('fEndAngle', _fEndAngle);
END_METHOD

METHOD PROTECTED SetMemberReference
VAR_INPUT
END_VAR
_aCenter.MakeReferenceTo(activeData.aCenter);
_fRadius.MakeReferenceTo(activeData.fRadius);
_fStartAngle.MakeReferenceTo(activeData.fStartAngle);
_fEndAngle.MakeReferenceTo(activeData.fEndAngle);
END_METHOD

METHOD PUBLIC Clone : I_Datatype
VAR
    pClone : POINTER TO _TcVnCircularArc;
END_VAR
pClone := __NEW(_TcVnCircularArc());
pClone^.Value := Value;
Clone := pClone^;
END_METHOD

PROPERTY PUBLIC Identifier : T_MAXSTRING
GET
Identifier := 'TcVnCircularArc';
END_GET
END_PROPERTY

METHOD PUBLIC MakeReferenceTo
VAR_INPUT
	ReferenceTarget : REFERENCE TO TcVnCircularArc;
END_VAR
activeData REF= ReferenceTarget;
SetMemberReference();
END_METHOD

METHOD TryMakeReferenceTo : BOOL
VAR_INPUT
	Target : I_Datatype;
END_VAR
VAR
	pTargetData : POINTER TO TcVnCircularArc;
END_VAR
IF NOT IsEquivalentTo(Target) THEN
	RETURN;
END_IF

pTargetData := Target.Address;
activeData REF= pTargetData^;
SetMemberReference();
TryMakeReferenceTo := TRUE;
END_METHOD

PROPERTY PUBLIC Value : REFERENCE TO TcVnCircularArc
GET
Value REF= activeData;
END_GET
END_PROPERTY

PROPERTY PUBLIC aCenter : REFERENCE TO _TcVnPoint2_REAL
GET
aCenter REF= _aCenter;
END_GET
END_PROPERTY

PROPERTY PUBLIC fEndAngle : REFERENCE TO _REAL
GET
fEndAngle REF= _fEndAngle;
END_GET
END_PROPERTY

PROPERTY PUBLIC fRadius : REFERENCE TO _REAL
GET
fRadius REF= _fRadius;
END_GET
END_PROPERTY

PROPERTY PUBLIC fStartAngle : REFERENCE TO _REAL
GET
fStartAngle REF= _fStartAngle;
END_GET
END_PROPERTY

END_FUNCTION_BLOCK

// Datatypes/Structs/_TcVnCodeGrades1D
{attribute 'linkalways'} 
{attribute 'no_explicit_call' := 'This FB is a CLASS and must be accessed using methods or properties'}
{attribute 'enable_dynamic_creation'}
FUNCTION_BLOCK _TcVnCodeGrades1D EXTENDS StructuredDatatypeBase
VAR
	localData : TcVnCodeGrades1D;
	activeData : REFERENCE TO TcVnCodeGrades1D REF= localData;
    _fDecode : _REAL(localdata.fDecode);
    _fSymbolContrast : _REAL(localdata.fSymbolContrast);
    _fMinReflectance : _REAL(localdata.fMinReflectance);
    _fMinEdgeContrast : _REAL(localdata.fMinEdgeContrast);
    _fModulation : _REAL(localdata.fModulation);
    _fDefects : _REAL(localdata.fDefects);
    _fDecodability : _REAL(localdata.fDecodability);
    _fOverall : _REAL(localdata.fOverall);
END_VAR

PROPERTY PUBLIC Address : PVOID
GET
Address := ADR(activeData);
END_GET
END_PROPERTY

METHOD PUBLIC ClearReference
VAR_INPUT
END_VAR
activeData REF= localData;
SetMemberReference();
END_METHOD

PROPERTY PUBLIC Size : UDINT
GET
Size := SIZEOF(activeData);
END_GET
END_PROPERTY

METHOD FB_init : BOOL
VAR_INPUT
	bInitRetains : BOOL; // if TRUE, the retain variables are initialized (warm start / cold start)
	bInCopyCode : BOOL;  // if TRUE, the instance afterwards gets moved into the copy code (online change)
END_VAR
SetMemberReference();
AddMember('fDecode', _fDecode);
AddMember('fSymbolContrast', _fSymbolContrast);
AddMember('fMinReflectance', _fMinReflectance);
AddMember('fMinEdgeContrast', _fMinEdgeContrast);
AddMember('fModulation', _fModulation);
AddMember('fDefects', _fDefects);
AddMember('fDecodability', _fDecodability);
AddMember('fOverall', _fOverall);
END_METHOD

METHOD PROTECTED SetMemberReference
VAR_INPUT
END_VAR
_fDecode.MakeReferenceTo(activeData.fDecode);
_fSymbolContrast.MakeReferenceTo(activeData.fSymbolContrast);
_fMinReflectance.MakeReferenceTo(activeData.fMinReflectance);
_fMinEdgeContrast.MakeReferenceTo(activeData.fMinEdgeContrast);
_fModulation.MakeReferenceTo(activeData.fModulation);
_fDefects.MakeReferenceTo(activeData.fDefects);
_fDecodability.MakeReferenceTo(activeData.fDecodability);
_fOverall.MakeReferenceTo(activeData.fOverall);
END_METHOD

METHOD PUBLIC Clone : I_Datatype
VAR
    pClone : POINTER TO _TcVnCodeGrades1D;
END_VAR
pClone := __NEW(_TcVnCodeGrades1D());
pClone^.Value := Value;
Clone := pClone^;
END_METHOD

PROPERTY PUBLIC Identifier : T_MAXSTRING
GET
Identifier := 'TcVnCodeGrades1D';
END_GET
END_PROPERTY

METHOD PUBLIC MakeReferenceTo
VAR_INPUT
	ReferenceTarget : REFERENCE TO TcVnCodeGrades1D;
END_VAR
activeData REF= ReferenceTarget;
SetMemberReference();
END_METHOD

METHOD TryMakeReferenceTo : BOOL
VAR_INPUT
	Target : I_Datatype;
END_VAR
VAR
	pTargetData : POINTER TO TcVnCodeGrades1D;
END_VAR
IF NOT IsEquivalentTo(Target) THEN
	RETURN;
END_IF

pTargetData := Target.Address;
activeData REF= pTargetData^;
SetMemberReference();
TryMakeReferenceTo := TRUE;
END_METHOD

PROPERTY PUBLIC Value : REFERENCE TO TcVnCodeGrades1D
GET
Value REF= activeData;
END_GET
END_PROPERTY

PROPERTY PUBLIC fDecodability : REFERENCE TO _REAL
GET
fDecodability REF= _fDecodability;
END_GET
END_PROPERTY

PROPERTY PUBLIC fDecode : REFERENCE TO _REAL
GET
fDecode REF= _fDecode;
END_GET
END_PROPERTY

PROPERTY PUBLIC fDefects : REFERENCE TO _REAL
GET
fDefects REF= _fDefects;
END_GET
END_PROPERTY

PROPERTY PUBLIC fMinEdgeContrast : REFERENCE TO _REAL
GET
fMinEdgeContrast REF= _fMinEdgeContrast;
END_GET
END_PROPERTY

PROPERTY PUBLIC fMinReflectance : REFERENCE TO _REAL
GET
fMinReflectance REF= _fMinReflectance;
END_GET
END_PROPERTY

PROPERTY PUBLIC fModulation : REFERENCE TO _REAL
GET
fModulation REF= _fModulation;
END_GET
END_PROPERTY

PROPERTY PUBLIC fOverall : REFERENCE TO _REAL
GET
fOverall REF= _fOverall;
END_GET
END_PROPERTY

PROPERTY PUBLIC fSymbolContrast : REFERENCE TO _REAL
GET
fSymbolContrast REF= _fSymbolContrast;
END_GET
END_PROPERTY

END_FUNCTION_BLOCK

// Datatypes/Structs/_TcVnCodeGradesDM
{attribute 'linkalways'} 
{attribute 'no_explicit_call' := 'This FB is a CLASS and must be accessed using methods or properties'}
{attribute 'enable_dynamic_creation'}
FUNCTION_BLOCK _TcVnCodeGradesDM EXTENDS StructuredDatatypeBase
VAR
	localData : TcVnCodeGradesDM;
	activeData : REFERENCE TO TcVnCodeGradesDM REF= localData;
    _nDecode : _USINT(localdata.nDecode);
    _nSymbolContrast : _USINT(localdata.nSymbolContrast);
    _nModulation : _USINT(localdata.nModulation);
    _nReflectanceMargin : _USINT(localdata.nReflectanceMargin);
    _nFixedPatternDamage : _USINT(localdata.nFixedPatternDamage);
    _nAxialNonuniformity : _USINT(localdata.nAxialNonuniformity);
    _nGridNonuniformity : _USINT(localdata.nGridNonuniformity);
    _nUnusedErrorCorrection : _USINT(localdata.nUnusedErrorCorrection);
    _nOverall : _USINT(localdata.nOverall);
END_VAR

PROPERTY PUBLIC Address : PVOID
GET
Address := ADR(activeData);
END_GET
END_PROPERTY

METHOD PUBLIC ClearReference
VAR_INPUT
END_VAR
activeData REF= localData;
SetMemberReference();
END_METHOD

PROPERTY PUBLIC Size : UDINT
GET
Size := SIZEOF(activeData);
END_GET
END_PROPERTY

METHOD FB_init : BOOL
VAR_INPUT
	bInitRetains : BOOL; // if TRUE, the retain variables are initialized (warm start / cold start)
	bInCopyCode : BOOL;  // if TRUE, the instance afterwards gets moved into the copy code (online change)
END_VAR
SetMemberReference();
AddMember('nDecode', _nDecode);
AddMember('nSymbolContrast', _nSymbolContrast);
AddMember('nModulation', _nModulation);
AddMember('nReflectanceMargin', _nReflectanceMargin);
AddMember('nFixedPatternDamage', _nFixedPatternDamage);
AddMember('nAxialNonuniformity', _nAxialNonuniformity);
AddMember('nGridNonuniformity', _nGridNonuniformity);
AddMember('nUnusedErrorCorrection', _nUnusedErrorCorrection);
AddMember('nOverall', _nOverall);
END_METHOD

METHOD PROTECTED SetMemberReference
VAR_INPUT
END_VAR
_nDecode.MakeReferenceTo(activeData.nDecode);
_nSymbolContrast.MakeReferenceTo(activeData.nSymbolContrast);
_nModulation.MakeReferenceTo(activeData.nModulation);
_nReflectanceMargin.MakeReferenceTo(activeData.nReflectanceMargin);
_nFixedPatternDamage.MakeReferenceTo(activeData.nFixedPatternDamage);
_nAxialNonuniformity.MakeReferenceTo(activeData.nAxialNonuniformity);
_nGridNonuniformity.MakeReferenceTo(activeData.nGridNonuniformity);
_nUnusedErrorCorrection.MakeReferenceTo(activeData.nUnusedErrorCorrection);
_nOverall.MakeReferenceTo(activeData.nOverall);
END_METHOD

METHOD PUBLIC Clone : I_Datatype
VAR
    pClone : POINTER TO _TcVnCodeGradesDM;
END_VAR
pClone := __NEW(_TcVnCodeGradesDM());
pClone^.Value := Value;
Clone := pClone^;
END_METHOD

PROPERTY PUBLIC Identifier : T_MAXSTRING
GET
Identifier := 'TcVnCodeGradesDM';
END_GET
END_PROPERTY

METHOD PUBLIC MakeReferenceTo
VAR_INPUT
	ReferenceTarget : REFERENCE TO TcVnCodeGradesDM;
END_VAR
activeData REF= ReferenceTarget;
SetMemberReference();
END_METHOD

METHOD TryMakeReferenceTo : BOOL
VAR_INPUT
	Target : I_Datatype;
END_VAR
VAR
	pTargetData : POINTER TO TcVnCodeGradesDM;
END_VAR
IF NOT IsEquivalentTo(Target) THEN
	RETURN;
END_IF

pTargetData := Target.Address;
activeData REF= pTargetData^;
SetMemberReference();
TryMakeReferenceTo := TRUE;
END_METHOD

PROPERTY PUBLIC Value : REFERENCE TO TcVnCodeGradesDM
GET
Value REF= activeData;
END_GET
END_PROPERTY

PROPERTY PUBLIC nAxialNonuniformity : REFERENCE TO _USINT
GET
nAxialNonuniformity REF= _nAxialNonuniformity;
END_GET
END_PROPERTY

PROPERTY PUBLIC nDecode : REFERENCE TO _USINT
GET
nDecode REF= _nDecode;
END_GET
END_PROPERTY

PROPERTY PUBLIC nFixedPatternDamage : REFERENCE TO _USINT
GET
nFixedPatternDamage REF= _nFixedPatternDamage;
END_GET
END_PROPERTY

PROPERTY PUBLIC nGridNonuniformity : REFERENCE TO _USINT
GET
nGridNonuniformity REF= _nGridNonuniformity;
END_GET
END_PROPERTY

PROPERTY PUBLIC nModulation : REFERENCE TO _USINT
GET
nModulation REF= _nModulation;
END_GET
END_PROPERTY

PROPERTY PUBLIC nOverall : REFERENCE TO _USINT
GET
nOverall REF= _nOverall;
END_GET
END_PROPERTY

PROPERTY PUBLIC nReflectanceMargin : REFERENCE TO _USINT
GET
nReflectanceMargin REF= _nReflectanceMargin;
END_GET
END_PROPERTY

PROPERTY PUBLIC nSymbolContrast : REFERENCE TO _USINT
GET
nSymbolContrast REF= _nSymbolContrast;
END_GET
END_PROPERTY

PROPERTY PUBLIC nUnusedErrorCorrection : REFERENCE TO _USINT
GET
nUnusedErrorCorrection REF= _nUnusedErrorCorrection;
END_GET
END_PROPERTY

END_FUNCTION_BLOCK

// Datatypes/Structs/_TcVnCodeGradesQR
{attribute 'linkalways'} 
{attribute 'no_explicit_call' := 'This FB is a CLASS and must be accessed using methods or properties'}
{attribute 'enable_dynamic_creation'}
FUNCTION_BLOCK _TcVnCodeGradesQR EXTENDS StructuredDatatypeBase
VAR
	localData : TcVnCodeGradesQR;
	activeData : REFERENCE TO TcVnCodeGradesQR REF= localData;
    _nDecode : _USINT(localdata.nDecode);
    _nSymbolContrast : _USINT(localdata.nSymbolContrast);
    _nModulation : _USINT(localdata.nModulation);
    _nReflectanceMargin : _USINT(localdata.nReflectanceMargin);
    _nFixedPatternDamage : _USINT(localdata.nFixedPatternDamage);
    _nAxialNonuniformity : _USINT(localdata.nAxialNonuniformity);
    _nGridNonuniformity : _USINT(localdata.nGridNonuniformity);
    _nUnusedErrorCorrection : _USINT(localdata.nUnusedErrorCorrection);
    _nFormatInfo : _USINT(localdata.nFormatInfo);
    _nVersionInfo : _USINT(localdata.nVersionInfo);
    _nOverall : _USINT(localdata.nOverall);
END_VAR

PROPERTY PUBLIC Address : PVOID
GET
Address := ADR(activeData);
END_GET
END_PROPERTY

METHOD PUBLIC ClearReference
VAR_INPUT
END_VAR
activeData REF= localData;
SetMemberReference();
END_METHOD

PROPERTY PUBLIC Size : UDINT
GET
Size := SIZEOF(activeData);
END_GET
END_PROPERTY

METHOD FB_init : BOOL
VAR_INPUT
	bInitRetains : BOOL; // if TRUE, the retain variables are initialized (warm start / cold start)
	bInCopyCode : BOOL;  // if TRUE, the instance afterwards gets moved into the copy code (online change)
END_VAR
SetMemberReference();
AddMember('nDecode', _nDecode);
AddMember('nSymbolContrast', _nSymbolContrast);
AddMember('nModulation', _nModulation);
AddMember('nReflectanceMargin', _nReflectanceMargin);
AddMember('nFixedPatternDamage', _nFixedPatternDamage);
AddMember('nAxialNonuniformity', _nAxialNonuniformity);
AddMember('nGridNonuniformity', _nGridNonuniformity);
AddMember('nUnusedErrorCorrection', _nUnusedErrorCorrection);
AddMember('nFormatInfo', _nFormatInfo);
AddMember('nVersionInfo', _nVersionInfo);
AddMember('nOverall', _nOverall);
END_METHOD

METHOD PROTECTED SetMemberReference
VAR_INPUT
END_VAR
_nDecode.MakeReferenceTo(activeData.nDecode);
_nSymbolContrast.MakeReferenceTo(activeData.nSymbolContrast);
_nModulation.MakeReferenceTo(activeData.nModulation);
_nReflectanceMargin.MakeReferenceTo(activeData.nReflectanceMargin);
_nFixedPatternDamage.MakeReferenceTo(activeData.nFixedPatternDamage);
_nAxialNonuniformity.MakeReferenceTo(activeData.nAxialNonuniformity);
_nGridNonuniformity.MakeReferenceTo(activeData.nGridNonuniformity);
_nUnusedErrorCorrection.MakeReferenceTo(activeData.nUnusedErrorCorrection);
_nFormatInfo.MakeReferenceTo(activeData.nFormatInfo);
_nVersionInfo.MakeReferenceTo(activeData.nVersionInfo);
_nOverall.MakeReferenceTo(activeData.nOverall);
END_METHOD

METHOD PUBLIC Clone : I_Datatype
VAR
    pClone : POINTER TO _TcVnCodeGradesQR;
END_VAR
pClone := __NEW(_TcVnCodeGradesQR());
pClone^.Value := Value;
Clone := pClone^;
END_METHOD

PROPERTY PUBLIC Identifier : T_MAXSTRING
GET
Identifier := 'TcVnCodeGradesQR';
END_GET
END_PROPERTY

METHOD PUBLIC MakeReferenceTo
VAR_INPUT
	ReferenceTarget : REFERENCE TO TcVnCodeGradesQR;
END_VAR
activeData REF= ReferenceTarget;
SetMemberReference();
END_METHOD

METHOD TryMakeReferenceTo : BOOL
VAR_INPUT
	Target : I_Datatype;
END_VAR
VAR
	pTargetData : POINTER TO TcVnCodeGradesQR;
END_VAR
IF NOT IsEquivalentTo(Target) THEN
	RETURN;
END_IF

pTargetData := Target.Address;
activeData REF= pTargetData^;
SetMemberReference();
TryMakeReferenceTo := TRUE;
END_METHOD

PROPERTY PUBLIC Value : REFERENCE TO TcVnCodeGradesQR
GET
Value REF= activeData;
END_GET
END_PROPERTY

PROPERTY PUBLIC nAxialNonuniformity : REFERENCE TO _USINT
GET
nAxialNonuniformity REF= _nAxialNonuniformity;
END_GET
END_PROPERTY

PROPERTY PUBLIC nDecode : REFERENCE TO _USINT
GET
nDecode REF= _nDecode;
END_GET
END_PROPERTY

PROPERTY PUBLIC nFixedPatternDamage : REFERENCE TO _USINT
GET
nFixedPatternDamage REF= _nFixedPatternDamage;
END_GET
END_PROPERTY

PROPERTY PUBLIC nFormatInfo : REFERENCE TO _USINT
GET
nFormatInfo REF= _nFormatInfo;
END_GET
END_PROPERTY

PROPERTY PUBLIC nGridNonuniformity : REFERENCE TO _USINT
GET
nGridNonuniformity REF= _nGridNonuniformity;
END_GET
END_PROPERTY

PROPERTY PUBLIC nModulation : REFERENCE TO _USINT
GET
nModulation REF= _nModulation;
END_GET
END_PROPERTY

PROPERTY PUBLIC nOverall : REFERENCE TO _USINT
GET
nOverall REF= _nOverall;
END_GET
END_PROPERTY

PROPERTY PUBLIC nReflectanceMargin : REFERENCE TO _USINT
GET
nReflectanceMargin REF= _nReflectanceMargin;
END_GET
END_PROPERTY

PROPERTY PUBLIC nSymbolContrast : REFERENCE TO _USINT
GET
nSymbolContrast REF= _nSymbolContrast;
END_GET
END_PROPERTY

PROPERTY PUBLIC nUnusedErrorCorrection : REFERENCE TO _USINT
GET
nUnusedErrorCorrection REF= _nUnusedErrorCorrection;
END_GET
END_PROPERTY

PROPERTY PUBLIC nVersionInfo : REFERENCE TO _USINT
GET
nVersionInfo REF= _nVersionInfo;
END_GET
END_PROPERTY

END_FUNCTION_BLOCK

// Datatypes/Structs/_TcVnMoments
{attribute 'linkalways'} 
{attribute 'no_explicit_call' := 'This FB is a CLASS and must be accessed using methods or properties'}
{attribute 'enable_dynamic_creation'}
FUNCTION_BLOCK _TcVnMoments EXTENDS StructuredDatatypeBase
VAR
	localData : TcVnMoments;
	activeData : REFERENCE TO TcVnMoments REF= localData;
    _fM00 : _LREAL(localdata.fM00);
    _fM01 : _LREAL(localdata.fM01);
    _fM02 : _LREAL(localdata.fM02);
    _fM03 : _LREAL(localdata.fM03);
    _fM10 : _LREAL(localdata.fM10);
    _fM11 : _LREAL(localdata.fM11);
    _fM12 : _LREAL(localdata.fM12);
    _fM20 : _LREAL(localdata.fM20);
    _fM21 : _LREAL(localdata.fM21);
    _fM30 : _LREAL(localdata.fM30);
    _fMu02 : _LREAL(localdata.fMu02);
    _fMu03 : _LREAL(localdata.fMu03);
    _fMu11 : _LREAL(localdata.fMu11);
    _fMu12 : _LREAL(localdata.fMu12);
    _fMu20 : _LREAL(localdata.fMu20);
    _fMu21 : _LREAL(localdata.fMu21);
    _fMu30 : _LREAL(localdata.fMu30);
    _fNu02 : _LREAL(localdata.fNu02);
    _fNu03 : _LREAL(localdata.fNu03);
    _fNu11 : _LREAL(localdata.fNu11);
    _fNu12 : _LREAL(localdata.fNu12);
    _fNu20 : _LREAL(localdata.fNu20);
    _fNu21 : _LREAL(localdata.fNu21);
    _fNu30 : _LREAL(localdata.fNu30);
END_VAR

PROPERTY PUBLIC Address : PVOID
GET
Address := ADR(activeData);
END_GET
END_PROPERTY

METHOD PUBLIC ClearReference
VAR_INPUT
END_VAR
activeData REF= localData;
SetMemberReference();
END_METHOD

PROPERTY PUBLIC Size : UDINT
GET
Size := SIZEOF(activeData);
END_GET
END_PROPERTY

METHOD FB_init : BOOL
VAR_INPUT
	bInitRetains : BOOL; // if TRUE, the retain variables are initialized (warm start / cold start)
	bInCopyCode : BOOL;  // if TRUE, the instance afterwards gets moved into the copy code (online change)
END_VAR
SetMemberReference();
AddMember('fM00', _fM00);
AddMember('fM01', _fM01);
AddMember('fM02', _fM02);
AddMember('fM03', _fM03);
AddMember('fM10', _fM10);
AddMember('fM11', _fM11);
AddMember('fM12', _fM12);
AddMember('fM20', _fM20);
AddMember('fM21', _fM21);
AddMember('fM30', _fM30);
AddMember('fMu02', _fMu02);
AddMember('fMu03', _fMu03);
AddMember('fMu11', _fMu11);
AddMember('fMu12', _fMu12);
AddMember('fMu20', _fMu20);
AddMember('fMu21', _fMu21);
AddMember('fMu30', _fMu30);
AddMember('fNu02', _fNu02);
AddMember('fNu03', _fNu03);
AddMember('fNu11', _fNu11);
AddMember('fNu12', _fNu12);
AddMember('fNu20', _fNu20);
AddMember('fNu21', _fNu21);
AddMember('fNu30', _fNu30);
END_METHOD

METHOD PROTECTED SetMemberReference
VAR_INPUT
END_VAR
_fM00.MakeReferenceTo(activeData.fM00);
_fM01.MakeReferenceTo(activeData.fM01);
_fM02.MakeReferenceTo(activeData.fM02);
_fM03.MakeReferenceTo(activeData.fM03);
_fM10.MakeReferenceTo(activeData.fM10);
_fM11.MakeReferenceTo(activeData.fM11);
_fM12.MakeReferenceTo(activeData.fM12);
_fM20.MakeReferenceTo(activeData.fM20);
_fM21.MakeReferenceTo(activeData.fM21);
_fM30.MakeReferenceTo(activeData.fM30);
_fMu02.MakeReferenceTo(activeData.fMu02);
_fMu03.MakeReferenceTo(activeData.fMu03);
_fMu11.MakeReferenceTo(activeData.fMu11);
_fMu12.MakeReferenceTo(activeData.fMu12);
_fMu20.MakeReferenceTo(activeData.fMu20);
_fMu21.MakeReferenceTo(activeData.fMu21);
_fMu30.MakeReferenceTo(activeData.fMu30);
_fNu02.MakeReferenceTo(activeData.fNu02);
_fNu03.MakeReferenceTo(activeData.fNu03);
_fNu11.MakeReferenceTo(activeData.fNu11);
_fNu12.MakeReferenceTo(activeData.fNu12);
_fNu20.MakeReferenceTo(activeData.fNu20);
_fNu21.MakeReferenceTo(activeData.fNu21);
_fNu30.MakeReferenceTo(activeData.fNu30);
END_METHOD

METHOD PUBLIC Clone : I_Datatype
VAR
    pClone : POINTER TO _TcVnMoments;
END_VAR
pClone := __NEW(_TcVnMoments());
pClone^.Value := Value;
Clone := pClone^;
END_METHOD

PROPERTY PUBLIC Identifier : T_MAXSTRING
GET
Identifier := 'TcVnMoments';
END_GET
END_PROPERTY

METHOD PUBLIC MakeReferenceTo
VAR_INPUT
	ReferenceTarget : REFERENCE TO TcVnMoments;
END_VAR
activeData REF= ReferenceTarget;
SetMemberReference();
END_METHOD

METHOD TryMakeReferenceTo : BOOL
VAR_INPUT
	Target : I_Datatype;
END_VAR
VAR
	pTargetData : POINTER TO TcVnMoments;
END_VAR
IF NOT IsEquivalentTo(Target) THEN
	RETURN;
END_IF

pTargetData := Target.Address;
activeData REF= pTargetData^;
SetMemberReference();
TryMakeReferenceTo := TRUE;
END_METHOD

PROPERTY PUBLIC Value : REFERENCE TO TcVnMoments
GET
Value REF= activeData;
END_GET
END_PROPERTY

PROPERTY PUBLIC fM00 : REFERENCE TO _LREAL
GET
fM00 REF= _fM00;
END_GET
END_PROPERTY

PROPERTY PUBLIC fM01 : REFERENCE TO _LREAL
GET
fM01 REF= _fM01;
END_GET
END_PROPERTY

PROPERTY PUBLIC fM02 : REFERENCE TO _LREAL
GET
fM02 REF= _fM02;
END_GET
END_PROPERTY

PROPERTY PUBLIC fM03 : REFERENCE TO _LREAL
GET
fM03 REF= _fM03;
END_GET
END_PROPERTY

PROPERTY PUBLIC fM10 : REFERENCE TO _LREAL
GET
fM10 REF= _fM10;
END_GET
END_PROPERTY

PROPERTY PUBLIC fM11 : REFERENCE TO _LREAL
GET
fM11 REF= _fM11;
END_GET
END_PROPERTY

PROPERTY PUBLIC fM12 : REFERENCE TO _LREAL
GET
fM12 REF= _fM12;
END_GET
END_PROPERTY

PROPERTY PUBLIC fM20 : REFERENCE TO _LREAL
GET
fM20 REF= _fM20;
END_GET
END_PROPERTY

PROPERTY PUBLIC fM21 : REFERENCE TO _LREAL
GET
fM21 REF= _fM21;
END_GET
END_PROPERTY

PROPERTY PUBLIC fM30 : REFERENCE TO _LREAL
GET
fM30 REF= _fM30;
END_GET
END_PROPERTY

PROPERTY PUBLIC fMu02 : REFERENCE TO _LREAL
GET
fMu02 REF= _fMu02;
END_GET
END_PROPERTY

PROPERTY PUBLIC fMu03 : REFERENCE TO _LREAL
GET
fMu03 REF= _fMu03;
END_GET
END_PROPERTY

PROPERTY PUBLIC fMu11 : REFERENCE TO _LREAL
GET
fMu11 REF= _fMu11;
END_GET
END_PROPERTY

PROPERTY PUBLIC fMu12 : REFERENCE TO _LREAL
GET
fMu12 REF= _fMu12;
END_GET
END_PROPERTY

PROPERTY PUBLIC fMu20 : REFERENCE TO _LREAL
GET
fMu20 REF= _fMu20;
END_GET
END_PROPERTY

PROPERTY PUBLIC fMu21 : REFERENCE TO _LREAL
GET
fMu21 REF= _fMu21;
END_GET
END_PROPERTY

PROPERTY PUBLIC fMu30 : REFERENCE TO _LREAL
GET
fMu30 REF= _fMu30;
END_GET
END_PROPERTY

PROPERTY PUBLIC fNu02 : REFERENCE TO _LREAL
GET
fNu02 REF= _fNu02;
END_GET
END_PROPERTY

PROPERTY PUBLIC fNu03 : REFERENCE TO _LREAL
GET
fNu03 REF= _fNu03;
END_GET
END_PROPERTY

PROPERTY PUBLIC fNu11 : REFERENCE TO _LREAL
GET
fNu11 REF= _fNu11;
END_GET
END_PROPERTY

PROPERTY PUBLIC fNu12 : REFERENCE TO _LREAL
GET
fNu12 REF= _fNu12;
END_GET
END_PROPERTY

PROPERTY PUBLIC fNu20 : REFERENCE TO _LREAL
GET
fNu20 REF= _fNu20;
END_GET
END_PROPERTY

PROPERTY PUBLIC fNu21 : REFERENCE TO _LREAL
GET
fNu21 REF= _fNu21;
END_GET
END_PROPERTY

PROPERTY PUBLIC fNu30 : REFERENCE TO _LREAL
GET
fNu30 REF= _fNu30;
END_GET
END_PROPERTY

END_FUNCTION_BLOCK

// Datatypes/Structs/_TcVnParamsAGAST
{attribute 'linkalways'} 
{attribute 'no_explicit_call' := 'This FB is a CLASS and must be accessed using methods or properties'}
{attribute 'enable_dynamic_creation'}
FUNCTION_BLOCK _TcVnParamsAGAST EXTENDS StructuredDatatypeBase
VAR
	localData : TcVnParamsAGAST;
	activeData : REFERENCE TO TcVnParamsAGAST REF= localData;
	_nThreshold : _DINT(localData.nThreshold);
    _bNonMaxSuppression : _BOOL(localData.bNonMaxSuppression);
	_eType : _ETcVnKeypointDetectionTypeAGAST(localData.eType);
END_VAR

PROPERTY PUBLIC Address : PVOID
GET
Address := ADR(activeData);
END_GET
END_PROPERTY

METHOD PUBLIC ClearReference
VAR_INPUT
END_VAR
activeData REF= localData;
SetMemberReference();
END_METHOD

PROPERTY PUBLIC Size : UDINT
GET
Size := SIZEOF(activeData);
END_GET
END_PROPERTY

METHOD FB_init : BOOL
VAR_INPUT
	bInitRetains : BOOL; // if TRUE, the retain variables are initialized (warm start / cold start)
	bInCopyCode : BOOL;  // if TRUE, the instance afterwards gets moved into the copy code (online change)
END_VAR
SetMemberReference();
AddMember('nThreshold',_nThreshold);
AddMember('bNonMaxSuppression',_bNonMaxSuppression );
AddMember('eType',_eType);
END_METHOD

METHOD PROTECTED SetMemberReference
VAR_INPUT
END_VAR
_nThreshold.MakeReferenceTo(activeData.nThreshold);
_bNonMaxSuppression.MakeReferenceTo(activeData.bNonMaxSuppression);
_eType.MakeReferenceTo(activeData.eType);
END_METHOD

METHOD PUBLIC Clone : I_Datatype
VAR
    pClone : POINTER TO _TcVnParamsAGAST;
END_VAR
pClone := __NEW(_TcVnParamsAGAST());
pClone^.Value := Value;
Clone := pClone^;
END_METHOD

PROPERTY PUBLIC Identifier : T_MAXSTRING
GET
Identifier := 'TcVnParamsAGAST';
END_GET
END_PROPERTY

METHOD PUBLIC MakeReferenceTo
VAR_INPUT
	ReferenceTarget : REFERENCE TO TcVnParamsAGAST;
END_VAR
activeData REF= ReferenceTarget;
SetMemberReference();
END_METHOD

METHOD TryMakeReferenceTo : BOOL
VAR_INPUT
	Target : I_Datatype;
END_VAR
VAR
	pTargetData : POINTER TO TcVnParamsAGAST;
END_VAR
IF NOT IsEquivalentTo(Target) THEN
	RETURN;
END_IF

pTargetData := Target.Address;
activeData REF= pTargetData^;
SetMemberReference();
TryMakeReferenceTo := TRUE;
END_METHOD

PROPERTY PUBLIC Value : REFERENCE TO TcVnParamsAGAST
GET
Value REF= activeData;
END_GET
END_PROPERTY

PROPERTY PUBLIC bNonMaxSuppression : REFERENCE TO _BOOL
GET
bNonMaxSuppression REF= _bNonMaxSuppression;
END_GET
END_PROPERTY

PROPERTY PUBLIC eType : REFERENCE TO _ETcVnKeypointDetectionTypeAGAST
GET
eType REF= _eType;
END_GET
END_PROPERTY

PROPERTY PUBLIC nThreshold : REFERENCE TO _DINT
GET
nThreshold REF= _nThreshold;
END_GET
END_PROPERTY

END_FUNCTION_BLOCK

// Datatypes/Structs/_TcVnParamsAKAZE
{attribute 'linkalways'} 
{attribute 'no_explicit_call' := 'This FB is a CLASS and must be accessed using methods or properties'}
{attribute 'enable_dynamic_creation'}
FUNCTION_BLOCK _TcVnParamsAKAZE EXTENDS StructuredDatatypeBase
VAR
	localData : TcVnParamsAKAZE;
	activeData : REFERENCE TO TcVnParamsAKAZE REF= localData;
    _eDescrType     : _ETcVnFeatureDescriptorTypeAKAZE(localdata.eDescrType);
    _nDescrSize     : _UDINT(localdata.nDescrSize);
    _nDescrChannels : _UDINT(localdata.nDescrChannels);
    _fThreshold     : _REAL(localdata.fThreshold);
    _nOctaves       : _UDINT(localdata.nOctaves);
    _nOctaveLayers  : _UDINT(localdata.nOctaveLayers);
    _eDiffusivity   : _ETcVnDiffusivityTypeKAZE(localdata.eDiffusivity);
END_VAR

PROPERTY PUBLIC Address : PVOID
GET
Address := ADR(activeData);
END_GET
END_PROPERTY

METHOD PUBLIC ClearReference
VAR_INPUT
END_VAR
activeData REF= localData;
SetMemberReference();
END_METHOD

PROPERTY PUBLIC Size : UDINT
GET
Size := SIZEOF(activeData);
END_GET
END_PROPERTY

METHOD FB_init : BOOL
VAR_INPUT
	bInitRetains : BOOL; // if TRUE, the retain variables are initialized (warm start / cold start)
	bInCopyCode : BOOL;  // if TRUE, the instance afterwards gets moved into the copy code (online change)
END_VAR
SetMemberReference();
AddMember('eDescrType', _eDescrType);
AddMember('nDescrSize', _nDescrSize);
AddMember('nDescrChannels', _nDescrChannels);
AddMember('fThreshold', _fThreshold);
AddMember('nOctaves', _nOctaves);
AddMember('nOctaveLayers', _nOctaveLayers);
AddMember('eDiffusivity', _eDiffusivity);
END_METHOD

METHOD PROTECTED SetMemberReference
VAR_INPUT
END_VAR
_eDescrType.MakeReferenceTo(activeData.eDescrType);
_nDescrSize.MakeReferenceTo(activeData.nDescrSize);
_nDescrChannels.MakeReferenceTo(activeData.nDescrChannels);
_fThreshold.MakeReferenceTo(activeData.fThreshold);
_nOctaves.MakeReferenceTo(activeData.nOctaves);
_nOctaveLayers.MakeReferenceTo(activeData.nOctaveLayers);
_eDiffusivity.MakeReferenceTo(activeData.eDiffusivity);
END_METHOD

METHOD PUBLIC Clone : I_Datatype
VAR
    pClone : POINTER TO _TcVnParamsAKAZE;
END_VAR
pClone := __NEW(_TcVnParamsAKAZE());
pClone^.Value := Value;
Clone := pClone^;
END_METHOD

PROPERTY PUBLIC Identifier : T_MAXSTRING
GET
Identifier := 'TcVnParamsAKAZE';
END_GET
END_PROPERTY

METHOD PUBLIC MakeReferenceTo
VAR_INPUT
	ReferenceTarget : REFERENCE TO TcVnParamsAKAZE;
END_VAR
activeData REF= ReferenceTarget;
SetMemberReference();
END_METHOD

METHOD TryMakeReferenceTo : BOOL
VAR_INPUT
	Target : I_Datatype;
END_VAR
VAR
	pTargetData : POINTER TO TcVnParamsAKAZE;
END_VAR
IF NOT IsEquivalentTo(Target) THEN
	RETURN;
END_IF

pTargetData := Target.Address;
activeData REF= pTargetData^;
SetMemberReference();
TryMakeReferenceTo := TRUE;
END_METHOD

PROPERTY PUBLIC Value : REFERENCE TO TcVnParamsAKAZE
GET
Value REF= activeData;
END_GET
END_PROPERTY

PROPERTY PUBLIC eDescrType : REFERENCE TO _ETcVnFeatureDescriptorTypeAKAZE
GET
eDescrType REF= _eDescrType;
END_GET
END_PROPERTY

PROPERTY PUBLIC eDiffusivity : REFERENCE TO _ETcVnDiffusivityTypeKAZE
GET
eDiffusivity REF= _eDiffusivity;
END_GET
END_PROPERTY

PROPERTY PUBLIC fThreshold : REFERENCE TO _REAL
GET
fThreshold REF= _fThreshold;
END_GET
END_PROPERTY

PROPERTY PUBLIC nDescrChannels : REFERENCE TO _UDINT
GET
nDescrChannels REF= _nDescrChannels;
END_GET
END_PROPERTY

PROPERTY PUBLIC nDescrSize : REFERENCE TO _UDINT
GET
nDescrSize REF= _nDescrSize;
END_GET
END_PROPERTY

PROPERTY PUBLIC nOctaveLayers : REFERENCE TO _UDINT
GET
nOctaveLayers REF= _nOctaveLayers;
END_GET
END_PROPERTY

PROPERTY PUBLIC nOctaves : REFERENCE TO _UDINT
GET
nOctaves REF= _nOctaves;
END_GET
END_PROPERTY

END_FUNCTION_BLOCK

// Datatypes/Structs/_TcVnParamsBlobDetection
{attribute 'linkalways'} 
{attribute 'no_explicit_call' := 'This FB is a CLASS and must be accessed using methods or properties'}
{attribute 'enable_dynamic_creation'}
FUNCTION_BLOCK _TcVnParamsBlobDetection EXTENDS StructuredDatatypeBase
VAR
	localData : TcVnParamsBlobDetection;
	activeData : REFERENCE TO TcVnParamsBlobDetection REF= localData;
    _bFilterByArea         : _BOOL(localdata.bFilterByArea);
    _bFilterByCircularity  : _BOOL(localdata.bFilterByCircularity);
    _bFilterByConvexity    : _BOOL(localdata.bFilterByConvexity);
    _bFilterByEccentricity : _BOOL(localdata.bFilterByEccentricity);
    _bFilterByInertiaRatio : _BOOL(localdata.bFilterByInertiaRatio);
    _fMinArea              : _REAL(localdata.fMinArea);
    _fMaxArea              : _REAL(localdata.fMaxArea);
    _fMinCircularity       : _REAL(localdata.fMinCircularity);
    _fMaxCircularity       : _REAL(localdata.fMaxCircularity);
    _fMinConvexity         : _REAL(localdata.fMinConvexity);
    _fMaxConvexity         : _REAL(localdata.fMaxConvexity);
    _fMinEccentricity      : _REAL(localdata.fMinEccentricity);
    _fMaxEccentricity      : _REAL(localdata.fMaxEccentricity);
    _fMinInertiaRatio      : _REAL(localdata.fMinInertiaRatio);
    _fMaxInertiaRatio      : _REAL(localdata.fMaxInertiaRatio);
    _eThresholdType        : _ETcVnThresholdType(localdata.eThresholdType);
    _fMinThreshold         : _REAL(localdata.fMinThreshold);
    _fMaxThreshold         : _REAL(localdata.fMaxThreshold);
    _fThresholdStep        : _REAL(localdata.fThresholdStep);
    _fMinBlobDistance      : _REAL(localdata.fMinBlobDistance);
    _nMinRepeatability     : _UDINT(localdata.nMinRepeatability);
    _eBlobCombination      : _ETcVnBlobCombination(localdata.eBlobCombination);
    _bExcludeBorderBlobs   : _BOOL(localdata.bExcludeBorderBlobs);
END_VAR

PROPERTY PUBLIC Address : PVOID
GET
Address := ADR(activeData);
END_GET
END_PROPERTY

METHOD PUBLIC ClearReference
VAR_INPUT
END_VAR
activeData REF= localData;
SetMemberReference();
END_METHOD

PROPERTY PUBLIC Size : UDINT
GET
Size := SIZEOF(activeData);
END_GET
END_PROPERTY

METHOD FB_init : BOOL
VAR_INPUT
	bInitRetains : BOOL; // if TRUE, the retain variables are initialized (warm start / cold start)
	bInCopyCode : BOOL;  // if TRUE, the instance afterwards gets moved into the copy code (online change)
END_VAR
SetMemberReference();
AddMember('bFilterByArea', _bFilterByArea);
AddMember('bFilterByCircularity', _bFilterByCircularity);
AddMember('bFilterByConvexity', _bFilterByConvexity);
AddMember('bFilterByEccentricity', _bFilterByEccentricity);
AddMember('bFilterByInertiaRatio', _bFilterByInertiaRatio);
AddMember('fMinArea', _fMinArea);
AddMember('fMaxArea', _fMaxArea);
AddMember('fMinCircularity', _fMinCircularity);
AddMember('fMaxCircularity', _fMaxCircularity);
AddMember('fMinConvexity', _fMinConvexity);
AddMember('fMaxConvexity', _fMaxConvexity);
AddMember('fMinEccentricity', _fMinEccentricity);
AddMember('fMaxEccentricity', _fMaxEccentricity);
AddMember('fMinInertiaRatio', _fMinInertiaRatio);
AddMember('fMaxInertiaRatio', _fMaxInertiaRatio);
AddMember('eThresholdType', _eThresholdType);
AddMember('fMinThreshold', _fMinThreshold);
AddMember('fMaxThreshold', _fMaxThreshold);
AddMember('fThresholdStep',  _fThresholdStep);
AddMember('fMinBlobDistance', _fMinBlobDistance);
AddMember('nMinRepeatability', _nMinRepeatability);
AddMember('eBlobCombination', _eBlobCombination);
AddMember('bExcludeBorderBlobs', _bExcludeBorderBlobs);
END_METHOD

METHOD PROTECTED SetMemberReference
VAR_INPUT
END_VAR
_bFilterByArea.MakeReferenceTo(activeData.bFilterByArea);
_bFilterByCircularity.MakeReferenceTo(activeData.bFilterByCircularity);
_bFilterByConvexity.MakeReferenceTo(activeData.bFilterByConvexity);
_bFilterByEccentricity.MakeReferenceTo(activeData.bFilterByEccentricity);
_bFilterByInertiaRatio.MakeReferenceTo(activeData.bFilterByInertiaRatio);
_fMinArea.MakeReferenceTo(activeData.fMinArea);
_fMaxArea.MakeReferenceTo(activeData.fMaxArea);
_fMinCircularity.MakeReferenceTo(activeData.fMinCircularity);
_fMaxCircularity.MakeReferenceTo(activeData.fMaxCircularity);
_fMinConvexity.MakeReferenceTo(activeData.fMinConvexity);
_fMaxConvexity.MakeReferenceTo(activeData.fMaxConvexity);
_fMinEccentricity.MakeReferenceTo(activeData.fMinEccentricity);
_fMaxEccentricity.MakeReferenceTo(activeData.fMaxEccentricity);
_fMinInertiaRatio.MakeReferenceTo(activeData.fMinInertiaRatio);
_fMaxInertiaRatio.MakeReferenceTo(activeData.fMaxInertiaRatio);
_eThresholdType.MakeReferenceTo(activeData.eThresholdType);
_fMinThreshold.MakeReferenceTo(activeData.fMinThreshold);
_fMaxThreshold.MakeReferenceTo(activeData.fMaxThreshold);
_fThresholdStep.MakeReferenceTo(activeData.fThresholdStep);
_fMinBlobDistance.MakeReferenceTo(activeData.fMinBlobDistance);
_nMinRepeatability.MakeReferenceTo(activeData.nMinRepeatability);
_eBlobCombination.MakeReferenceTo(activeData.eBlobCombination);
_bExcludeBorderBlobs.MakeReferenceTo(activeData.bExcludeBorderBlobs);
END_METHOD

METHOD PUBLIC Clone : I_Datatype
VAR
    pClone : POINTER TO _TcVnParamsBlobDetection;
END_VAR
pClone := __NEW(_TcVnParamsBlobDetection());
pClone^.Value := Value;
Clone := pClone^;
END_METHOD

PROPERTY PUBLIC Identifier : T_MAXSTRING
GET
Identifier := 'TcVnParamsBlobDetection';
END_GET
END_PROPERTY

METHOD PUBLIC MakeReferenceTo
VAR_INPUT
	ReferenceTarget : REFERENCE TO TcVnParamsBlobDetection;
END_VAR
activeData REF= ReferenceTarget;
SetMemberReference();
END_METHOD

METHOD TryMakeReferenceTo : BOOL
VAR_INPUT
	Target : I_Datatype;
END_VAR
VAR
	pTargetData : POINTER TO TcVnParamsBlobDetection;
END_VAR
IF NOT IsEquivalentTo(Target) THEN
	RETURN;
END_IF

pTargetData := Target.Address;
activeData REF= pTargetData^;
SetMemberReference();
TryMakeReferenceTo := TRUE;
END_METHOD

PROPERTY PUBLIC Value : REFERENCE TO TcVnParamsBlobDetection
GET
Value REF= activeData;
END_GET
END_PROPERTY

PROPERTY PUBLIC bExcludeBorderBlobs : REFERENCE TO _BOOL
GET
bExcludeBorderBlobs REF= _bExcludeBorderBlobs;
END_GET
END_PROPERTY

PROPERTY PUBLIC bFilterByArea : REFERENCE TO _BOOL
GET
bFilterByArea REF= _bFilterByArea;
END_GET
END_PROPERTY

PROPERTY PUBLIC bFilterByCircularity : REFERENCE TO _BOOL
GET
bFilterByCircularity REF= _bFilterByCircularity;
END_GET
END_PROPERTY

PROPERTY PUBLIC bFilterByConvexity : REFERENCE TO _BOOL
GET
bFilterByConvexity REF= _bFilterByConvexity;
END_GET
END_PROPERTY

PROPERTY PUBLIC bFilterByEccentricity : REFERENCE TO _BOOL
GET
bFilterByEccentricity REF= _bFilterByEccentricity;
END_GET
END_PROPERTY

PROPERTY PUBLIC bFilterByInertiaRatio : REFERENCE TO _BOOL
GET
bFilterByInertiaRatio REF= _bFilterByInertiaRatio;
END_GET
END_PROPERTY

PROPERTY PUBLIC eBlobCombination : REFERENCE TO _ETcVnBlobCombination
GET
eBlobCombination REF= _eBlobCombination;
END_GET
END_PROPERTY

PROPERTY PUBLIC eThresholdType : REFERENCE TO _ETcVnThresholdType
GET
eThresholdType REF= _eThresholdType;
END_GET
END_PROPERTY

PROPERTY PUBLIC fMaxArea : REFERENCE TO _REAL
GET
fMaxArea REF= _fMaxArea;
END_GET
END_PROPERTY

PROPERTY PUBLIC fMaxCircularity : REFERENCE TO _REAL
GET
fMaxCircularity REF= _fMaxCircularity;
END_GET
END_PROPERTY

PROPERTY PUBLIC fMaxConvexity : REFERENCE TO _REAL
GET
fMaxConvexity REF= _fMaxConvexity;
END_GET
END_PROPERTY

PROPERTY PUBLIC fMaxEccentricity : REFERENCE TO _REAL
GET
fMaxEccentricity REF= _fMaxEccentricity;
END_GET
END_PROPERTY

PROPERTY PUBLIC fMaxInertiaRatio : REFERENCE TO _REAL
GET
fMaxInertiaRatio REF= _fMaxInertiaRatio;
END_GET
END_PROPERTY

PROPERTY PUBLIC fMaxThreshold : REFERENCE TO _REAL
GET
fMaxThreshold REF= _fMaxThreshold;
END_GET
END_PROPERTY

PROPERTY PUBLIC fMinArea : REFERENCE TO _REAL
GET
fMinArea REF= _fMinArea;
END_GET
END_PROPERTY

PROPERTY PUBLIC fMinBlobDistance : REFERENCE TO _REAL
GET
fMinBlobDistance REF= _fMinBlobDistance;
END_GET
END_PROPERTY

PROPERTY PUBLIC fMinCircularity : REFERENCE TO _REAL
GET
fMinCircularity REF= _fMinCircularity;
END_GET
END_PROPERTY

PROPERTY PUBLIC fMinConvexity : REFERENCE TO _REAL
GET
fMinConvexity REF= _fMinConvexity;
END_GET
END_PROPERTY

PROPERTY PUBLIC fMinEccentricity : REFERENCE TO _REAL
GET
fMinEccentricity REF= _fMinEccentricity;
END_GET
END_PROPERTY

PROPERTY PUBLIC fMinInertiaRatio : REFERENCE TO _REAL
GET
fMinInertiaRatio REF= _fMinInertiaRatio;
END_GET
END_PROPERTY

PROPERTY PUBLIC fMinThreshold : REFERENCE TO _REAL
GET
fMinThreshold REF= _fMinThreshold;
END_GET
END_PROPERTY

PROPERTY PUBLIC fThresholdStep : REFERENCE TO _REAL
GET
fThresholdStep REF= _fThresholdStep;
END_GET
END_PROPERTY

PROPERTY PUBLIC nMinRepeatability : REFERENCE TO _UDINT
GET
nMinRepeatability REF= _nMinRepeatability;
END_GET
END_PROPERTY

END_FUNCTION_BLOCK

// Datatypes/Structs/_TcVnParamsBRISK
{attribute 'linkalways'} 
{attribute 'no_explicit_call' := 'This FB is a CLASS and must be accessed using methods or properties'}
{attribute 'enable_dynamic_creation'}
FUNCTION_BLOCK _TcVnParamsBRISK EXTENDS StructuredDatatypeBase
VAR
	localData : TcVnParamsBRISK;
	activeData : REFERENCE TO TcVnParamsBRISK REF= localData;
	_nThreshold : _DINT(localData.nThreshold);
	_nOctaves : _UDINT(localData.nOctaves);
	_fPatternScale : _REAL(localData.fPatternScale);
END_VAR

PROPERTY PUBLIC Address : PVOID
GET
Address := ADR(activeData);
END_GET
END_PROPERTY

METHOD PUBLIC ClearReference
VAR_INPUT
END_VAR
activeData REF= localData;
SetMemberReference();
END_METHOD

PROPERTY PUBLIC Size : UDINT
GET
Size := SIZEOF(activeData);
END_GET
END_PROPERTY

METHOD FB_init : BOOL
VAR_INPUT
	bInitRetains : BOOL; // if TRUE, the retain variables are initialized (warm start / cold start)
	bInCopyCode : BOOL;  // if TRUE, the instance afterwards gets moved into the copy code (online change)
END_VAR
SetMemberReference();
AddMember('nThreshold', _nThreshold);
AddMember('nOctaves', _nOctaves);
AddMember('fPatternScale', _fPatternScale);
END_METHOD

METHOD PROTECTED SetMemberReference
VAR_INPUT
END_VAR
_nThreshold.MakeReferenceTo(activeData.nThreshold);
_nOctaves.MakeReferenceTo(activeData.nOctaves);
_fPatternScale.MakeReferenceTo(activeData.fPatternScale);
END_METHOD

METHOD PUBLIC Clone : I_Datatype
VAR
    pClone : POINTER TO _TcVnParamsBRISK;
END_VAR
pClone := __NEW(_TcVnParamsBRISK());
pClone^.Value := Value;
Clone := pClone^;
END_METHOD

PROPERTY PUBLIC Identifier : T_MAXSTRING
GET
Identifier := 'TcVnParamsBRISK';
END_GET
END_PROPERTY

METHOD PUBLIC MakeReferenceTo
VAR_INPUT
	ReferenceTarget : REFERENCE TO TcVnParamsBRISK;
END_VAR
activeData REF= ReferenceTarget;
SetMemberReference();
END_METHOD

METHOD TryMakeReferenceTo : BOOL
VAR_INPUT
	Target : I_Datatype;
END_VAR
VAR
	pTargetData : POINTER TO TcVnParamsBRISK;
END_VAR
IF NOT IsEquivalentTo(Target) THEN
	RETURN;
END_IF

pTargetData := Target.Address;
activeData REF= pTargetData^;
SetMemberReference();
TryMakeReferenceTo := TRUE;
END_METHOD

PROPERTY PUBLIC Value : REFERENCE TO TcVnParamsBRISK
GET
Value REF= activeData;
END_GET
END_PROPERTY

PROPERTY PUBLIC fPatternScale : REFERENCE TO _REAL
GET
fPatternScale REF= _fPatternScale;
END_GET
END_PROPERTY

PROPERTY PUBLIC nOctaves : REFERENCE TO _UDINT
GET
nOctaves REF= _nOctaves;
END_GET
END_PROPERTY

PROPERTY PUBLIC nThreshold : REFERENCE TO _DINT
GET
nThreshold REF= _nThreshold;
END_GET
END_PROPERTY

METHOD PUBLIC TryDeserializeFrom : BOOL
VAR_INPUT
    Deserializer : I_Deserializer;
    Feedback : I_DeserializerFeedback;
END_VAR
VAR
    membersEnumerator : I_DeserializerObjectForwardEnumerator;
    member : I_Datatype;
    memberName : T_MAXSTRING;
END_VAR
// Map the legacy member name without advertising or serializing it twice.
membersEnumerator := Deserializer.GetObjectEnumerator();
WHILE membersEnumerator.MoveNext() DO
    memberName := membersEnumerator.Key;
    IF memberName = 'fPatternScale ' THEN
        memberName := 'fPatternScale';
    END_IF
    IF Members.TryGetMemberByName(memberName, member) THEN
        IF NOT member.TryDeserializeFrom(membersEnumerator.Current, Feedback) THEN
            membersEnumerator.Dispose();
            RETURN;
        END_IF
    END_IF
END_WHILE
membersEnumerator.Dispose();
TryDeserializeFrom := TRUE;
END_METHOD

END_FUNCTION_BLOCK

// Datatypes/Structs/_TcVnParamsFAST
{attribute 'linkalways'} 
{attribute 'no_explicit_call' := 'This FB is a CLASS and must be accessed using methods or properties'}
{attribute 'enable_dynamic_creation'}
FUNCTION_BLOCK _TcVnParamsFAST EXTENDS StructuredDatatypeBase
VAR
	localData : TcVnParamsFAST;
	activeData : REFERENCE TO TcVnParamsFAST REF= localData;
	_nThreshold : _DINT(localData.nThreshold);
    _bNonMaxSuppression : _BOOL(localData.bNonMaxSuppression);
	_eType : _ETcVnKeypointDetectionTypeFAST(localData.eType);
END_VAR

PROPERTY PUBLIC Address : PVOID
GET
Address := ADR(activeData);
END_GET
END_PROPERTY

METHOD PUBLIC ClearReference
VAR_INPUT
END_VAR
activeData REF= localData;
SetMemberReference();
END_METHOD

PROPERTY PUBLIC Size : UDINT
GET
Size := SIZEOF(activeData);
END_GET
END_PROPERTY

METHOD FB_init : BOOL
VAR_INPUT
	bInitRetains : BOOL; // if TRUE, the retain variables are initialized (warm start / cold start)
	bInCopyCode : BOOL;  // if TRUE, the instance afterwards gets moved into the copy code (online change)
END_VAR
SetMemberReference();
AddMember('nThreshold',_nThreshold);
AddMember('bNonMaxSuppression',_bNonMaxSuppression );
AddMember('eType',_eType);
END_METHOD

METHOD PROTECTED SetMemberReference
VAR_INPUT
END_VAR
_nThreshold.MakeReferenceTo(activeData.nThreshold);
_bNonMaxSuppression.MakeReferenceTo(activeData.bNonMaxSuppression);
_eType.MakeReferenceTo(activeData.eType);
END_METHOD

METHOD PUBLIC Clone : I_Datatype
VAR
    pClone : POINTER TO _TcVnParamsFAST;
END_VAR
pClone := __NEW(_TcVnParamsFAST());
pClone^.Value := Value;
Clone := pClone^;
END_METHOD

PROPERTY PUBLIC Identifier : T_MAXSTRING
GET
Identifier := 'TcVnParamsFAST';
END_GET
END_PROPERTY

METHOD PUBLIC MakeReferenceTo
VAR_INPUT
	ReferenceTarget : REFERENCE TO TcVnParamsFAST;
END_VAR
activeData REF= ReferenceTarget;
SetMemberReference();
END_METHOD

METHOD TryMakeReferenceTo : BOOL
VAR_INPUT
	Target : I_Datatype;
END_VAR
VAR
	pTargetData : POINTER TO TcVnParamsFAST;
END_VAR
IF NOT IsEquivalentTo(Target) THEN
	RETURN;
END_IF

pTargetData := Target.Address;
activeData REF= pTargetData^;
SetMemberReference();
TryMakeReferenceTo := TRUE;
END_METHOD

PROPERTY PUBLIC Value : REFERENCE TO TcVnParamsFAST
GET
Value REF= activeData;
END_GET
END_PROPERTY

PROPERTY PUBLIC bNonMaxSuppression : REFERENCE TO _BOOL
GET
bNonMaxSuppression REF= _bNonMaxSuppression;
END_GET
END_PROPERTY

PROPERTY PUBLIC eType : REFERENCE TO _ETcVnKeypointDetectionTypeFAST
GET
eType REF= _eType;
END_GET
END_PROPERTY

PROPERTY PUBLIC nThreshold : REFERENCE TO _DINT
GET
nThreshold REF= _nThreshold;
END_GET
END_PROPERTY

END_FUNCTION_BLOCK

// Datatypes/Structs/_TcVnParamsFindRois
{attribute 'linkalways'}
{attribute 'no_explicit_call' := 'This FB is a CLASS and must be accessed using methods or properties'}
{attribute 'enable_dynamic_creation'}
FUNCTION_BLOCK _TcVnParamsFindRois EXTENDS StructuredDatatypeBase
VAR
    localData : TcVnParamsFindRois := (stRoiSize := (nWidth := 416, nHeight := 416), fMinDensity := 0.2, fDetectionScaleFactor := 0.25, fMaxOversizeFraction := 1.0);
    activeData : REFERENCE TO TcVnParamsFindRois REF= localData;
    _stRoiSize : _TcVnSize2_DINT;
    _fMinDensity : _LREAL(localData.fMinDensity);
    _fDetectionScaleFactor : _LREAL(localData.fDetectionScaleFactor);
    _fMaxOversizeFraction : _LREAL(localData.fMaxOversizeFraction);
END_VAR

PROPERTY PUBLIC Address : PVOID
GET
Address := ADR(activeData);
END_GET
END_PROPERTY

METHOD PUBLIC ClearReference
VAR_INPUT
END_VAR
activeData REF= localData;
SetMemberReference();
END_METHOD

PROPERTY PUBLIC Size : UDINT
GET
Size := SIZEOF(activeData);
END_GET
END_PROPERTY

METHOD FB_init : BOOL
VAR_INPUT
	bInitRetains : BOOL; // if TRUE, the retain variables are initialized (warm start / cold start)
	bInCopyCode : BOOL;  // if TRUE, the instance afterwards gets moved into the copy code (online change)
END_VAR
SetMemberReference();
AddMember('stRoiSize', _stRoiSize);
AddMember('fMinDensity', _fMinDensity);
AddMember('fDetectionScaleFactor', _fDetectionScaleFactor);
AddMember('fMaxOversizeFraction', _fMaxOversizeFraction);
END_METHOD

METHOD PROTECTED SetMemberReference
VAR_INPUT
END_VAR
_stRoiSize.MakeReferenceTo(activeData.stRoiSize);
_fMinDensity.MakeReferenceTo(activeData.fMinDensity);
_fDetectionScaleFactor.MakeReferenceTo(activeData.fDetectionScaleFactor);
_fMaxOversizeFraction.MakeReferenceTo(activeData.fMaxOversizeFraction);
END_METHOD

METHOD PUBLIC Clone : I_Datatype
VAR
    pClone : POINTER TO _TcVnParamsFindRois;
END_VAR
pClone := __NEW(_TcVnParamsFindRois);
IF pClone = 0 THEN
    RETURN;
END_IF
pClone^.TryCopyFrom(THIS^);
Clone := pClone^;
END_METHOD

PROPERTY PUBLIC Identifier : T_MAXSTRING
GET
Identifier := 'TcVnParamsFindRois';
END_GET
END_PROPERTY

METHOD PUBLIC MakeReferenceTo
VAR_INPUT
	ReferenceTarget : REFERENCE TO TcVnParamsFindRois;
END_VAR
activeData REF= ReferenceTarget;
SetMemberReference();
END_METHOD

METHOD TryMakeReferenceTo : BOOL
VAR_INPUT
	Target : I_Datatype;
END_VAR
VAR
	pTargetData : POINTER TO TcVnParamsFindRois;
END_VAR
IF NOT IsEquivalentTo(Target) THEN
	RETURN;
END_IF

pTargetData := Target.Address;
activeData REF= pTargetData^;
SetMemberReference();
TryMakeReferenceTo := TRUE;
END_METHOD

PROPERTY PUBLIC Value : REFERENCE TO TcVnParamsFindRois
GET
Value REF= activeData;
END_GET
END_PROPERTY

PROPERTY PUBLIC fDetectionScaleFactor : REFERENCE TO _LREAL
GET
fDetectionScaleFactor REF= _fDetectionScaleFactor;
END_GET
END_PROPERTY

PROPERTY PUBLIC fMaxOversizeFraction : REFERENCE TO _LREAL
GET
fMaxOversizeFraction REF= _fMaxOversizeFraction;
END_GET
END_PROPERTY

PROPERTY PUBLIC fMinDensity : REFERENCE TO _LREAL
GET
fMinDensity REF= _fMinDensity;
END_GET
END_PROPERTY

PROPERTY PUBLIC stRoiSize : REFERENCE TO _TcVnSize2_DINT
GET
stRoiSize REF= _stRoiSize;
END_GET
END_PROPERTY

END_FUNCTION_BLOCK

// Datatypes/Structs/_TcVnSize2_DINT
{attribute 'linkalways'}
{attribute 'no_explicit_call' := 'This FB is a CLASS and must be accessed using methods or properties'}
{attribute 'enable_dynamic_creation'}
FUNCTION_BLOCK _TcVnSize2_DINT EXTENDS StructuredDatatypeBase
VAR
    localData : TcVnSize2_DINT;
    activeData : REFERENCE TO TcVnSize2_DINT REF= localData;
    _nWidth : _DINT(localData.nWidth);
    _nHeight : _DINT(localData.nHeight);
END_VAR

PROPERTY PUBLIC Address : PVOID
GET
Address := ADR(activeData);
END_GET
END_PROPERTY

METHOD PUBLIC ClearReference
VAR_INPUT
END_VAR
activeData REF= localData;
SetMemberReference();
END_METHOD

PROPERTY PUBLIC Size : UDINT
GET
Size := SIZEOF(activeData);
END_GET
END_PROPERTY

METHOD FB_init : BOOL
VAR_INPUT
	bInitRetains : BOOL; // if TRUE, the retain variables are initialized (warm start / cold start)
	bInCopyCode : BOOL;  // if TRUE, the instance afterwards gets moved into the copy code (online change)
END_VAR
SetMemberReference();
AddMember('nWidth', _nWidth);
AddMember('nHeight', _nHeight);
END_METHOD

METHOD PROTECTED SetMemberReference
VAR_INPUT
END_VAR
_nWidth.MakeReferenceTo(activeData.nWidth);
_nHeight.MakeReferenceTo(activeData.nHeight);
END_METHOD

METHOD PUBLIC Clone : I_Datatype
VAR
    pClone : POINTER TO _TcVnSize2_DINT;
END_VAR
pClone := __NEW(_TcVnSize2_DINT);
IF pClone = 0 THEN
    RETURN;
END_IF
pClone^.TryCopyFrom(THIS^);
Clone := pClone^;
END_METHOD

PROPERTY PUBLIC Identifier : T_MAXSTRING
GET
Identifier := 'TcVnSize2_DINT';
END_GET
END_PROPERTY

METHOD PUBLIC MakeReferenceTo
VAR_INPUT
	ReferenceTarget : REFERENCE TO TcVnSize2_DINT;
END_VAR
activeData REF= ReferenceTarget;
SetMemberReference();
END_METHOD

METHOD TryMakeReferenceTo : BOOL
VAR_INPUT
	Target : I_Datatype;
END_VAR
VAR
	pTargetData : POINTER TO TcVnSize2_DINT;
END_VAR
IF NOT IsEquivalentTo(Target) THEN
	RETURN;
END_IF

pTargetData := Target.Address;
activeData REF= pTargetData^;
SetMemberReference();
TryMakeReferenceTo := TRUE;
END_METHOD

PROPERTY PUBLIC Value : REFERENCE TO TcVnSize2_DINT
GET
Value REF= activeData;
END_GET
END_PROPERTY

PROPERTY PUBLIC nHeight : REFERENCE TO _DINT
GET
nHeight REF= _nHeight;
END_GET
END_PROPERTY

PROPERTY PUBLIC nWidth : REFERENCE TO _DINT
GET
nWidth REF= _nWidth;
END_GET
END_PROPERTY

END_FUNCTION_BLOCK

// Datatypes/Structs/_TcVnParamsGFTT
{attribute 'linkalways'} 
{attribute 'no_explicit_call' := 'This FB is a CLASS and must be accessed using methods or properties'}
{attribute 'enable_dynamic_creation'}
FUNCTION_BLOCK _TcVnParamsGFTT EXTENDS StructuredDatatypeBase
VAR
	localData : TcVnParamsGFTT;
	activeData : REFERENCE TO TcVnParamsGFTT REF= localData;
	_nMaxCorners : _UDINT(localData.nMaxCorners);
    _fQualityLevel : _LREAL(localData.fQualityLevel);
	_fMinDistance : _LREAL(localData.fMinDistance);
	_nBlockSize : _UDINT(localData.nBlockSize);
	_bUseHarrisDetector : _BOOL(localData.bUseHarrisDetector);
	_fHarrisK : _LREAL(localData.fHarrisK);
END_VAR

PROPERTY PUBLIC Address : PVOID
GET
Address := ADR(activeData);
END_GET
END_PROPERTY

METHOD PUBLIC ClearReference
VAR_INPUT
END_VAR
activeData REF= localData;
SetMemberReference();
END_METHOD

PROPERTY PUBLIC Size : UDINT
GET
Size := SIZEOF(activeData);
END_GET
END_PROPERTY

METHOD FB_init : BOOL
VAR_INPUT
	bInitRetains : BOOL; // if TRUE, the retain variables are initialized (warm start / cold start)
	bInCopyCode : BOOL;  // if TRUE, the instance afterwards gets moved into the copy code (online change)
END_VAR
SetMemberReference();
AddMember('nMaxCorners', _nMaxCorners);
AddMember('fQualityLevel', _fQualityLevel);
AddMember('fMinDistance', _fMinDistance);
AddMember('nBlockSize', _nBlockSize);
AddMember('bUseHarrisDetector', _bUseHarrisDetector);
AddMember('fHarrisK', _fHarrisK);
END_METHOD

METHOD PROTECTED SetMemberReference
VAR_INPUT
END_VAR
_nMaxCorners.MakeReferenceTo(activeData.nMaxCorners);
_fQualityLevel.MakeReferenceTo(activeData.fQualityLevel);
_fMinDistance.MakeReferenceTo(activeData.fMinDistance);
_nBlockSize.MakeReferenceTo(activeData.nBlockSize);
_bUseHarrisDetector.MakeReferenceTo(activeData.bUseHarrisDetector);
_fHarrisK.MakeReferenceTo(activeData.fHarrisK);
END_METHOD

METHOD PUBLIC Clone : I_Datatype
VAR
    pClone : POINTER TO _TcVnParamsGFTT;
END_VAR
pClone := __NEW(_TcVnParamsGFTT());
pClone^.Value := Value;
Clone := pClone^;
END_METHOD

PROPERTY PUBLIC Identifier : T_MAXSTRING
GET
Identifier := 'TcVnParamsGFTT';
END_GET
END_PROPERTY

METHOD PUBLIC MakeReferenceTo
VAR_INPUT
	ReferenceTarget : REFERENCE TO TcVnParamsGFTT;
END_VAR
activeData REF= ReferenceTarget;
SetMemberReference();
END_METHOD

METHOD TryMakeReferenceTo : BOOL
VAR_INPUT
	Target : I_Datatype;
END_VAR
VAR
	pTargetData : POINTER TO TcVnParamsGFTT;
END_VAR
IF NOT IsEquivalentTo(Target) THEN
	RETURN;
END_IF

pTargetData := Target.Address;
activeData REF= pTargetData^;
SetMemberReference();
TryMakeReferenceTo := TRUE;
END_METHOD

PROPERTY PUBLIC Value : REFERENCE TO TcVnParamsGFTT
GET
Value REF= activeData;
END_GET
END_PROPERTY

PROPERTY PUBLIC bUseHarrisDetector : REFERENCE TO _BOOL
GET
bUseHarrisDetector REF= _bUseHarrisDetector;
END_GET
END_PROPERTY

PROPERTY PUBLIC fHarrisK : REFERENCE TO _LREAL
GET
fHarrisK REF= _fHarrisK;
END_GET
END_PROPERTY

PROPERTY PUBLIC fMinDistance : REFERENCE TO _LREAL
GET
fMinDistance REF= _fMinDistance;
END_GET
END_PROPERTY

PROPERTY PUBLIC fQualityLevel : REFERENCE TO _LREAL
GET
fQualityLevel REF= _fQualityLevel;
END_GET
END_PROPERTY

PROPERTY PUBLIC nBlockSize : REFERENCE TO _UDINT
GET
nBlockSize REF= _nBlockSize;
END_GET
END_PROPERTY

PROPERTY PUBLIC nMaxCorners : REFERENCE TO _UDINT
GET
nMaxCorners REF= _nMaxCorners;
END_GET
END_PROPERTY

END_FUNCTION_BLOCK

// Datatypes/Structs/_TcVnParamsKAZE
{attribute 'linkalways'} 
{attribute 'no_explicit_call' := 'This FB is a CLASS and must be accessed using methods or properties'}
{attribute 'enable_dynamic_creation'}
FUNCTION_BLOCK _TcVnParamsKAZE EXTENDS StructuredDatatypeBase
VAR
	localData : TcVnParamsKAZE;
	activeData : REFERENCE TO TcVnParamsKAZE REF= localData;
    _bExtended     : _BOOL(localdata.bExtended);
    _bUpright      : _BOOL(localdata.bUpright);
    _fThreshold    : _REAL(localdata.fThreshold);
    _nOctaves      : _UDINT(localdata.nOctaves);
    _nOctaveLayers : _UDINT(localdata.nOctaveLayers);
    _eDiffusivity  : _ETcVnDiffusivityTypeKAZE(localdata.eDiffusivity);
END_VAR

PROPERTY PUBLIC Address : PVOID
GET
Address := ADR(activeData);
END_GET
END_PROPERTY

METHOD PUBLIC ClearReference
VAR_INPUT
END_VAR
activeData REF= localData;
SetMemberReference();
END_METHOD

PROPERTY PUBLIC Size : UDINT
GET
Size := SIZEOF(activeData);
END_GET
END_PROPERTY

METHOD FB_init : BOOL
VAR_INPUT
	bInitRetains : BOOL; // if TRUE, the retain variables are initialized (warm start / cold start)
	bInCopyCode : BOOL;  // if TRUE, the instance afterwards gets moved into the copy code (online change)
END_VAR
SetMemberReference();
AddMember('bExtended', _bExtended);
AddMember('bUpright', _bUpright);
AddMember('fThreshold', _fThreshold);
AddMember('nOctaves', _nOctaves);
AddMember('nOctaveLayers', _nOctaveLayers);
AddMember('eDiffusivity', _eDiffusivity);
END_METHOD

METHOD PROTECTED SetMemberReference
VAR_INPUT
END_VAR
_bExtended.MakeReferenceTo(activeData.bExtended);
_bUpright.MakeReferenceTo(activeData.bUpright);
_fThreshold.MakeReferenceTo(activeData.fThreshold);
_nOctaves.MakeReferenceTo(activeData.nOctaves);
_nOctaveLayers.MakeReferenceTo(activeData.nOctaveLayers);
_eDiffusivity.MakeReferenceTo(activeData.eDiffusivity);
END_METHOD

METHOD PUBLIC Clone : I_Datatype
VAR
    pClone : POINTER TO _TcVnParamsKAZE;
END_VAR
pClone := __NEW(_TcVnParamsKAZE());
pClone^.Value := Value;
Clone := pClone^;
END_METHOD

PROPERTY PUBLIC Identifier : T_MAXSTRING
GET
Identifier := 'TcVnParamsKAZE';
END_GET
END_PROPERTY

METHOD PUBLIC MakeReferenceTo
VAR_INPUT
	ReferenceTarget : REFERENCE TO TcVnParamsKAZE;
END_VAR
activeData REF= ReferenceTarget;
SetMemberReference();
END_METHOD

METHOD TryMakeReferenceTo : BOOL
VAR_INPUT
	Target : I_Datatype;
END_VAR
VAR
	pTargetData : POINTER TO TcVnParamsKAZE;
END_VAR
IF NOT IsEquivalentTo(Target) THEN
	RETURN;
END_IF

pTargetData := Target.Address;
activeData REF= pTargetData^;
SetMemberReference();
TryMakeReferenceTo := TRUE;
END_METHOD

PROPERTY PUBLIC Value : REFERENCE TO TcVnParamsKAZE
GET
Value REF= activeData;
END_GET
END_PROPERTY

PROPERTY PUBLIC bExtended : REFERENCE TO _BOOL
GET
bExtended REF= _bExtended;
END_GET
END_PROPERTY

PROPERTY PUBLIC bUpright : REFERENCE TO _BOOL
GET
bUpright REF= _bUpright;
END_GET
END_PROPERTY

PROPERTY PUBLIC eDiffusivity : REFERENCE TO _ETcVnDiffusivityTypeKAZE
GET
eDiffusivity REF= _eDiffusivity;
END_GET
END_PROPERTY

PROPERTY PUBLIC fThreshold : REFERENCE TO _REAL
GET
fThreshold REF= _fThreshold;
END_GET
END_PROPERTY

PROPERTY PUBLIC nOctaveLayers : REFERENCE TO _UDINT
GET
nOctaveLayers REF= _nOctaveLayers;
END_GET
END_PROPERTY

PROPERTY PUBLIC nOctaves : REFERENCE TO _UDINT
GET
nOctaves REF= _nOctaves;
END_GET
END_PROPERTY

END_FUNCTION_BLOCK

// Datatypes/Structs/_TcVnParamsMSER
{attribute 'linkalways'} 
{attribute 'no_explicit_call' := 'This FB is a CLASS and must be accessed using methods or properties'}
{attribute 'enable_dynamic_creation'}
FUNCTION_BLOCK _TcVnParamsMSER EXTENDS StructuredDatatypeBase
VAR
	localData : TcVnParamsMSER;
	activeData : REFERENCE TO TcVnParamsMSER REF= localData;
	_nDelta : _DINT(localData.nDelta);
    _nMinArea : _UDINT(localData.nMinArea);
	_nMaxArea : _UDINT(localData.nMaxArea);
	_fMaxVariation : _LREAL(localData.fMaxVariation);
	_fMinDiversity : _LREAL(localData.fMinDiversity);
	_nMaxEvolution : _UDINT(localData.nMaxEvolution);
    _fAreaThreshold : _LREAL(localData.fAreaThreshold);
    _fMinMargin : _LREAL(localData.fMinMargin);
    _nEdgeBlurSize : _UDINT(localData.nEdgeBlurSize);
END_VAR

PROPERTY PUBLIC Address : PVOID
GET
Address := ADR(activeData);
END_GET
END_PROPERTY

METHOD PUBLIC ClearReference
VAR_INPUT
END_VAR
activeData REF= localData;
SetMemberReference();
END_METHOD

PROPERTY PUBLIC Size : UDINT
GET
Size := SIZEOF(activeData);
END_GET
END_PROPERTY

METHOD FB_init : BOOL
VAR_INPUT
	bInitRetains : BOOL; // if TRUE, the retain variables are initialized (warm start / cold start)
	bInCopyCode : BOOL;  // if TRUE, the instance afterwards gets moved into the copy code (online change)
END_VAR
SetMemberReference();
AddMember('nDelta', _nDelta);
AddMember('nMinArea', _nMinArea);
AddMember('nMaxArea', _nMaxArea);
AddMember('fMaxVariation', _fMaxVariation);
AddMember('fMinDiversity', _fMinDiversity);
AddMember('nMaxEvolution', _nMaxEvolution);
AddMember('fAreaThreshold', _fAreaThreshold);
AddMember('fMinMargin', _fMinMargin);
AddMember('nEdgeBlurSize', _nEdgeBlurSize);
END_METHOD

METHOD PROTECTED SetMemberReference
VAR_INPUT
END_VAR
_nDelta.MakeReferenceTo(activeData.nDelta);
_nMinArea.MakeReferenceTo(activeData.nMinArea);
_nMaxArea.MakeReferenceTo(activeData.nMaxArea);
_fMaxVariation.MakeReferenceTo(activeData.fMaxVariation);
_fMinDiversity.MakeReferenceTo(activeData.fMinDiversity);
_nMaxEvolution.MakeReferenceTo(activeData.nMaxEvolution);
_fAreaThreshold.MakeReferenceTo(activeData.fAreaThreshold);
_fMinMargin.MakeReferenceTo(activeData.fMinMargin);
_nEdgeBlurSize.MakeReferenceTo(activeData.nEdgeBlurSize);
END_METHOD

METHOD PUBLIC Clone : I_Datatype
VAR
    pClone : POINTER TO _TcVnParamsMSER;
END_VAR
pClone := __NEW(_TcVnParamsMSER());
pClone^.Value := Value;
Clone := pClone^;
END_METHOD

PROPERTY PUBLIC Identifier : T_MAXSTRING
GET
Identifier := 'TcVnParamsMSER';
END_GET
END_PROPERTY

METHOD PUBLIC MakeReferenceTo
VAR_INPUT
	ReferenceTarget : REFERENCE TO TcVnParamsMSER;
END_VAR
activeData REF= ReferenceTarget;
SetMemberReference();
END_METHOD

METHOD TryMakeReferenceTo : BOOL
VAR_INPUT
	Target : I_Datatype;
END_VAR
VAR
	pTargetData : POINTER TO TcVnParamsMSER;
END_VAR
IF NOT IsEquivalentTo(Target) THEN
	RETURN;
END_IF

pTargetData := Target.Address;
activeData REF= pTargetData^;
SetMemberReference();
TryMakeReferenceTo := TRUE;
END_METHOD

PROPERTY PUBLIC Value : REFERENCE TO TcVnParamsMSER
GET
Value REF= activeData;
END_GET
END_PROPERTY

PROPERTY PUBLIC fAreaThreshold : REFERENCE TO _LREAL
GET
fAreaThreshold REF= _fAreaThreshold;
END_GET
END_PROPERTY

PROPERTY PUBLIC fMaxVariation : REFERENCE TO _LREAL
GET
fMaxVariation REF= _fMaxVariation;
END_GET
END_PROPERTY

PROPERTY PUBLIC fMinDiversity : REFERENCE TO _LREAL
GET
fMinDiversity REF= _fMinDiversity;
END_GET
END_PROPERTY

PROPERTY PUBLIC fMinMargin : REFERENCE TO _LREAL
GET
fMinMargin REF= _fMinMargin;
END_GET
END_PROPERTY

PROPERTY PUBLIC nDelta : REFERENCE TO _DINT
GET
nDelta REF= _nDelta;
END_GET
END_PROPERTY

PROPERTY PUBLIC nEdgeBlurSize : REFERENCE TO _UDINT
GET
nEdgeBlurSize REF= _nEdgeBlurSize;
END_GET
END_PROPERTY

PROPERTY PUBLIC nMaxArea : REFERENCE TO _UDINT
GET
nMaxArea REF= _nMaxArea;
END_GET
END_PROPERTY

PROPERTY PUBLIC nMaxEvolution : REFERENCE TO _UDINT
GET
nMaxEvolution REF= _nMaxEvolution;
END_GET
END_PROPERTY

PROPERTY PUBLIC nMinArea : REFERENCE TO _UDINT
GET
nMinArea REF= _nMinArea;
END_GET
END_PROPERTY

END_FUNCTION_BLOCK

// Datatypes/Structs/_TcVnParamsORB
{attribute 'linkalways'} 
{attribute 'no_explicit_call' := 'This FB is a CLASS and must be accessed using methods or properties'}
{attribute 'enable_dynamic_creation'}
FUNCTION_BLOCK _TcVnParamsORB EXTENDS StructuredDatatypeBase
VAR
	localData : TcVnParamsORB;
	activeData : REFERENCE TO TcVnParamsORB REF= localData;
    _nMaxPoints : _UDINT(localData.nMaxPoints);
    _fPyramidScale : _REAL(localData.fPyramidScale);
    _nPyramidLevels : _UDINT(localData.nPyramidLevels);
    _nEdgeThreshold : _UDINT(localData.nEdgeThreshold);
    _nFirstLevel : _UDINT(localData.nFirstLevel);
    _nBriefPoints : _UDINT(localData.nBriefPoints);
    _eScoreType : _ETcVnFeatureScoreTypeORB(localData.eScoreType);
    _nPatchSize : _UDINT(localData.nPatchSize);
    _nFastThreshold : _DINT(localData.nFastThreshold);
END_VAR

PROPERTY PUBLIC Address : PVOID
GET
Address := ADR(activeData);
END_GET
END_PROPERTY

METHOD PUBLIC ClearReference
VAR_INPUT
END_VAR
activeData REF= localData;
SetMemberReference();
END_METHOD

PROPERTY PUBLIC Size : UDINT
GET
Size := SIZEOF(activeData);
END_GET
END_PROPERTY

METHOD FB_init : BOOL
VAR_INPUT
	bInitRetains : BOOL; // if TRUE, the retain variables are initialized (warm start / cold start)
	bInCopyCode : BOOL;  // if TRUE, the instance afterwards gets moved into the copy code (online change)
END_VAR
SetMemberReference();
AddMember('nMaxPoints', _nMaxPoints);
AddMember('fPyramidScale', _fPyramidScale);
AddMember('nPyramidLevels', _nPyramidLevels);
AddMember('nEdgeThreshold', _nEdgeThreshold);
AddMember('nFirstLevel', _nFirstLevel);
AddMember('nBriefPoints', _nBriefPoints);
AddMember('eScoreType', _eScoreType);
AddMember('nPatchSize', _nPatchSize);
AddMember('nFastThreshold', _nFastThreshold);
END_METHOD

METHOD PROTECTED SetMemberReference
VAR_INPUT
END_VAR
_nMaxPoints.MakeReferenceTo(activeData.nMaxPoints);
_fPyramidScale.MakeReferenceTo(activeData.fPyramidScale);
_nPyramidLevels.MakeReferenceTo(activeData.nPyramidLevels);
_nEdgeThreshold.MakeReferenceTo(activeData.nEdgeThreshold);
_nFirstLevel.MakeReferenceTo(activeData.nFirstLevel);
_nBriefPoints.MakeReferenceTo(activeData.nBriefPoints);
_eScoreType.MakeReferenceTo(activeData.eScoreType);
_nPatchSize.MakeReferenceTo(activeData.nPatchSize);
_nFastThreshold.MakeReferenceTo(activeData.nFastThreshold);
END_METHOD

METHOD PUBLIC Clone : I_Datatype
VAR
    pClone : POINTER TO _TcVnParamsORB;
END_VAR
pClone := __NEW(_TcVnParamsORB());
pClone^.Value := Value;
Clone := pClone^;
END_METHOD

PROPERTY PUBLIC Identifier : T_MAXSTRING
GET
Identifier := 'TcVnParamsORB';
END_GET
END_PROPERTY

METHOD PUBLIC MakeReferenceTo
VAR_INPUT
	ReferenceTarget : REFERENCE TO TcVnParamsORB;
END_VAR
activeData REF= ReferenceTarget;
SetMemberReference();
END_METHOD

METHOD TryMakeReferenceTo : BOOL
VAR_INPUT
	Target : I_Datatype;
END_VAR
VAR
	pTargetData : POINTER TO TcVnParamsORB;
END_VAR
IF NOT IsEquivalentTo(Target) THEN
	RETURN;
END_IF

pTargetData := Target.Address;
activeData REF= pTargetData^;
SetMemberReference();
TryMakeReferenceTo := TRUE;
END_METHOD

PROPERTY PUBLIC Value : REFERENCE TO TcVnParamsORB
GET
Value REF= activeData;
END_GET
END_PROPERTY

PROPERTY PUBLIC eScoreType : REFERENCE TO _ETcVnFeatureScoreTypeORB
GET
eScoreType REF= _eScoreType;
END_GET
END_PROPERTY

PROPERTY PUBLIC fPyramidScale : REFERENCE TO _REAL
GET
fPyramidScale REF= _fPyramidScale;
END_GET
END_PROPERTY

PROPERTY PUBLIC nBriefPoints : REFERENCE TO _UDINT
GET
nBriefPoints REF= _nBriefPoints;
END_GET
END_PROPERTY

PROPERTY PUBLIC nEdgeThreshold : REFERENCE TO _UDINT
GET
nEdgeThreshold REF= _nEdgeThreshold;
END_GET
END_PROPERTY

PROPERTY PUBLIC nFastThreshold : REFERENCE TO _DINT
GET
nFastThreshold REF= _nFastThreshold;
END_GET
END_PROPERTY

PROPERTY PUBLIC nFirstLevel : REFERENCE TO _UDINT
GET
nFirstLevel REF= _nFirstLevel;
END_GET
END_PROPERTY

PROPERTY PUBLIC nMaxPoints : REFERENCE TO _UDINT
GET
nMaxPoints REF= _nMaxPoints;
END_GET
END_PROPERTY

PROPERTY PUBLIC nPatchSize : REFERENCE TO _UDINT
GET
nPatchSize REF= _nPatchSize;
END_GET
END_PROPERTY

PROPERTY PUBLIC nPyramidLevels : REFERENCE TO _UDINT
GET
nPyramidLevels REF= _nPyramidLevels;
END_GET
END_PROPERTY

END_FUNCTION_BLOCK

// Datatypes/Structs/_TcVnParamsSB
{attribute 'linkalways'} 
{attribute 'no_explicit_call' := 'This FB is a CLASS and must be accessed using methods or properties'}
{attribute 'enable_dynamic_creation'}
FUNCTION_BLOCK _TcVnParamsSB EXTENDS StructuredDatatypeBase
VAR
	localData : TcVnParamsSB;
	activeData : REFERENCE TO TcVnParamsSB REF= localData;
    _bFilterByArea         : _BOOL(localdata.bFilterByArea);
    _bFilterByCircularity  : _BOOL(localdata.bFilterByCircularity);
    _bFilterByColor        : _BOOL(localdata.bFilterByColor);
    _bFilterByConvexity    : _BOOL(localdata.bFilterByConvexity);
    _bFilterByInertia      : _BOOL(localdata.bFilterByInertia);
    _fMinArea              : _REAL(localdata.fMinArea);
    _fMaxArea              : _REAL(localdata.fMaxArea);
    _fMinCircularity       : _REAL(localdata.fMinCircularity);
    _fMaxCircularity       : _REAL(localdata.fMaxCircularity);
    _nBlobColor            : _USINT(localdata.nBlobColor);
    _fMinConvexity         : _REAL(localdata.fMinConvexity);
    _fMaxConvexity         : _REAL(localdata.fMaxConvexity);
    _fMinInertiaRatio      : _REAL(localdata.fMinInertiaRatio);
    _fMaxInertiaRatio      : _REAL(localdata.fMaxInertiaRatio);
    _fMinBlobDist          : _REAL(localdata.fMinBlobDist);
    _nMinRepeatability     : _UDINT(localdata.nMinRepeatability);
    _fMinThreshold         : _REAL(localdata.fMinThreshold);
    _fMaxThreshold         : _REAL(localdata.fMaxThreshold);
    _fThresholdStep        : _REAL(localdata.fThresholdStep);
END_VAR

PROPERTY PUBLIC Address : PVOID
GET
Address := ADR(activeData);
END_GET
END_PROPERTY

